LIN {X 0,Y 297.473,Z 181.693,A -85,B 0,C 180,E1 -16448.382,E2 -16448.382} C_VEL
LIN {X 0,Y 297.609,Z 178.436,A -85,B 0,C 180,E1 -16452.122,E2 -16452.122} C_VEL
LIN {X 0,Y 297.859,Z 175.705,A -85,B 0,C 180,E1 -16455.326,E2 -16455.326} C_VEL
LIN {X 0,Y 298.134,Z 175.347,A -85,B 0,C 180,E1 -16457.751,E2 -16457.751} C_VEL
LIN {X 0,Y 298.702,Z 175.277,A -85,B 0,C 180,E1 -16461.884,E2 -16461.884} C_VEL
LIN {X 0,Y 298.65,Z 175.283,A -85,B 0,C 180,E1 -16464.598,E2 -16464.598} C_VEL
LIN {X 0,Y 298.921,Z 175.249,A -85,B 0,C 180,E1 -16468.653,E2 -16468.653} C_VEL
LIN {X 0,Y 298.921,Z 175.247,A -85,B 0,C 180,E1 -16471.347,E2 -16471.347} C_VEL
LIN {X 0,Y 298.794,Z 175.264,A -85,B 0,C 180,E1 -16476.754,E2 -16476.754} C_VEL
LIN {X 0,Y 298.677,Z 175.281,A -85,B 0,C 180,E1 -16479.48,E2 -16479.48} C_VEL
LIN {X 0,Y 298.549,Z 175.299,A -85,B 0,C 180,E1 -16483.615,E2 -16483.615} C_VEL
LIN {X 0,Y 298.545,Z 175.295,A -85,B 0,C 180,E1 -16486.409,E2 -16486.409} C_VEL
LIN {X 0,Y 298.508,Z 175.304,A -85,B 0,C 180,E1 -16489.655,E2 -16489.655} C_VEL
LIN {X 0,Y 298.454,Z 175.31,A -85,B 0,C 180,E1 -16493.598,E2 -16493.598} C_VEL
LIN {X 0,Y 298.482,Z 175.3,A -85,B 0,C 180,E1 -16496.575,E2 -16496.575} C_VEL
LIN {X 0,Y 298.413,Z 175.314,A -85,B 0,C 180,E1 -16499.642,E2 -16499.642} C_VEL
LIN {X 0,Y 298.391,Z 175.315,A -85,B 0,C 180,E1 -16502.801,E2 -16502.801} C_VEL
LIN {X 0,Y 298.441,Z 175.307,A -85,B 0,C 180,E1 -16506.807,E2 -16506.807} C_VEL
LIN {X 0,Y 298.385,Z 175.319,A -85,B 0,C 180,E1 -16511.088,E2 -16511.088} C_VEL
LIN {X 0,Y 298.386,Z 175.318,A -85,B 0,C 180,E1 -16515.042,E2 -16515.042} C_VEL
LIN {X 0,Y 298.385,Z 175.316,A -85,B 0,C 180,E1 -16518.913,E2 -16518.913} C_VEL
LIN {X 0,Y 298.442,Z 175.309,A -85,B 0,C 180,E1 -16523.193,E2 -16523.193} C_VEL
LIN {X 0,Y 298.393,Z 175.314,A -85,B 0,C 180,E1 -16527.2,E2 -16527.2} C_VEL
LIN {X 0,Y 298.425,Z 175.311,A -85,B 0,C 180,E1 -16530.617,E2 -16530.617} C_VEL
LIN {X 0,Y 298.476,Z 175.301,A -85,B 0,C 180,E1 -16533.477,E2 -16533.477} C_VEL
LIN {X 0,Y 298.435,Z 175.312,A -85,B 0,C 180,E1 -16536.698,E2 -16536.698} C_VEL
LIN {X 0,Y 298.539,Z 175.296,A -85,B 0,C 180,E1 -16540.758,E2 -16540.758} C_VEL
LIN {X 0,Y 298.593,Z 175.286,A -85,B 0,C 180,E1 -16544.996,E2 -16544.996} C_VEL
LIN {X 0,Y 298.592,Z 175.288,A -85,B 0,C 180,E1 -16549.147,E2 -16549.147} C_VEL
LIN {X 0,Y 298.741,Z 175.272,A -85,B 0,C 180,E1 -16551.886,E2 -16551.886} C_VEL
LIN {X 0,Y 298.713,Z 175.271,A -85,B 0,C 180,E1 -16553.806,E2 -16553.806} C_VEL
LIN {X 0,Y 297.983,Z 175.364,A -85,B 0,C 180,E1 -16554.931,E2 -16554.931} C_VEL
LIN {X 0,Y 295.181,Z 175.711,A -85,B 0,C 180,E1 -16556.768,E2 -16556.768} C_VEL
LIN {X 0,Y 292.899,Z 175.999,A -85,B 0,C 180,E1 -16558.258,E2 -16558.258} C_VEL
LIN {X 0,Y 291.986,Z 176.11,A -85,B 0,C 180,E1 -16559.41,E2 -16559.41} C_VEL
LIN {X 0,Y 291.944,Z 176.117,A -85,B 0,C 180,E1 -16559.799,E2 -16559.799} C_VEL
LIN {X 0,Y 291.788,Z 176.136,A -85,B 0,C 180,E1 -16562.762,E2 -16562.762} C_VEL
LIN {X 0,Y 291.7,Z 176.146,A -85,B 0,C 180,E1 -16566.92,E2 -16566.92} C_VEL
LIN {X 0,Y 291.569,Z 176.164,A -85,B 0,C 180,E1 -16569.715,E2 -16569.715} C_VEL
LIN {X 0,Y 291.524,Z 176.172,A -85,B 0,C 180,E1 -16573.951,E2 -16573.951} C_VEL
LIN {X 0,Y 291.489,Z 176.172,A -85,B 0,C 180,E1 -16576.818,E2 -16576.818} C_VEL
LIN {X 0,Y 291.452,Z 176.18,A -85,B 0,C 180,E1 -16579.875,E2 -16579.875} C_VEL
LIN {X 0,Y 291.401,Z 176.185,A -85,B 0,C 180,E1 -16584.206,E2 -16584.206} C_VEL
LIN {X 0,Y 291.421,Z 176.186,A -85,B 0,C 180,E1 -16587.272,E2 -16587.272} C_VEL
LIN {X 0,Y 291.336,Z 176.193,A -85,B 0,C 180,E1 -16590.438,E2 -16590.438} C_VEL
LIN {X 0,Y 291.347,Z 176.194,A -85,B 0,C 180,E1 -16593.699,E2 -16593.699} C_VEL
LIN {X 0,Y 291.378,Z 176.192,A -85,B 0,C 180,E1 -16597.255,E2 -16597.255} C_VEL
LIN {X 0,Y 291.382,Z 176.234,A -85,B 0,C 180,E1 -16599.836,E2 -16599.836} C_VEL
LIN {X 0,Y 292.261,Z 181.111,A -85,B 0,C 180,E1 -16603.829,E2 -16603.829} C_VEL
LIN {X 0,Y 293.231,Z 186.36,A -85,B 0,C 180,E1 -16607.849,E2 -16607.849} C_VEL
LIN {X 0,Y 294.105,Z 191.57,A -85,B 0,C 180,E1 -16611.589,E2 -16611.589} C_VEL
LIN {X 0,Y 294.167,Z 194.116,A -85,B 0,C 180,E1 -16613.325,E2 -16613.325} C_VEL
LIN {X 0,Y 293.464,Z 199.141,A -85,B 0,C 180,E1 -16616.577,E2 -16616.577} C_VEL
LIN {X 0,Y 292.415,Z 205.473,A -85,B 0,C 180,E1 -16620.549,E2 -16620.549} C_VEL
LIN {X 0,Y 291.542,Z 211.574,A -85,B 0,C 180,E1 -16624.284,E2 -16624.284} C_VEL
LIN {X 0,Y 291.27,Z 214.004,A -85,B 0,C 180,E1 -16625.724,E2 -16625.724} C_VEL
LIN {X 0,Y 293.669,Z 227.805,A -85,B 0,C 180,E1 -16626.542,E2 -16626.542} C_VEL
LIN {X 0,Y 295.547,Z 241.488,A -85,B 0,C 180,E1 -16627.637,E2 -16627.637} C_VEL
LIN {X 0,Y 296.631,Z 253.134,A -85,B 0,C 180,E1 -16628.799,E2 -16628.799} C_VEL
LIN {X 0,Y 296.996,Z 262.647,A -85,B 0,C 180,E1 -16629.933,E2 -16629.933} C_VEL
LIN {X 0,Y 295.444,Z 272.588,A -85,B 0,C 180,E1 -16631.268,E2 -16631.268} C_VEL
LIN {X 0,Y 293.939,Z 283.435,A -85,B 0,C 180,E1 -16633.114,E2 -16633.114} C_VEL
LIN {X 0,Y 292.546,Z 292.482,A -85,B 0,C 180,E1 -16635.034,E2 -16635.034} C_VEL
LIN {X 0,Y 291.363,Z 300.313,A -85,B 0,C 180,E1 -16637.108,E2 -16637.108} C_VEL
LIN {X 0,Y 290.452,Z 307.494,A -85,B 0,C 180,E1 -16639.544,E2 -16639.544} C_VEL
LIN {X 0,Y 289.911,Z 312.271,A -85,B 0,C 180,E1 -16641.637,E2 -16641.637} C_VEL
LIN {X 0,Y 289.677,Z 316.494,A -85,B 0,C 180,E1 -16644.117,E2 -16644.117} C_VEL
LIN {X 0,Y 289.602,Z 318.523,A -85,B 0,C 180,E1 -16645.825,E2 -16645.825} C_VEL
LIN {X 0,Y 289.558,Z 319.73,A -85,B 0,C 180,E1 -16647.218,E2 -16647.218} C_VEL
LIN {X 0,Y 289.58,Z 320.506,A -85,B 0,C 180,E1 -16648.61,E2 -16648.61} C_VEL
LIN {X 0,Y 289.688,Z 320.856,A -85,B 0,C 180,E1 -16650,E2 -16650} C_VEL
LIN {X 0,Y 289.545,Z 320.344,A -85,B 0,C 180,E1 -16652.783,E2 -16652.783} C_VEL
LIN {X 0,Y 289.557,Z 319.479,A -85,B 0,C 180,E1 -16654.176,E2 -16654.176} C_VEL
LIN {X 0,Y 289.633,Z 317.927,A -85,B 0,C 180,E1 -16655.798,E2 -16655.798} C_VEL
LIN {X 0,Y 289.908,Z 314.345,A -85,B 0,C 180,E1 -16658.364,E2 -16658.364} C_VEL
LIN {X 0,Y 290.452,Z 310.262,A -85,B 0,C 180,E1 -16660.456,E2 -16660.456} C_VEL
LIN {X 0,Y 291.439,Z 304.066,A -85,B 0,C 180,E1 -16662.889,E2 -16662.889} C_VEL
LIN {X 0,Y 292.984,Z 296.118,A -85,B 0,C 180,E1 -16665.3,E2 -16665.3} C_VEL
LIN {X 0,Y 294.468,Z 288.574,A -85,B 0,C 180,E1 -16667.128,E2 -16667.128} C_VEL
LIN {X 0,Y 296.202,Z 278.852,A -85,B 0,C 180,E1 -16669.041,E2 -16669.041} C_VEL
LIN {X 0,Y 298.212,Z 268.241,A -85,B 0,C 180,E1 -16670.702,E2 -16670.702} C_VEL
LIN {X 0,Y 298.925,Z 263.295,A -85,B 0,C 180,E1 -16671.372,E2 -16671.372} C_VEL
LIN {X 0,Y 298.806,Z 251.482,A -85,B 0,C 180,E1 -16672.872,E2 -16672.872} C_VEL
LIN {X 0,Y 297.979,Z 239.718,A -85,B 0,C 180,E1 -16674.143,E2 -16674.143} C_VEL
LIN {X 0,Y 295.872,Z 227.27,A -85,B 0,C 180,E1 -16675.344,E2 -16675.344} C_VEL
LIN {X 0,Y 292.582,Z 214.464,A -85,B 0,C 180,E1 -16676.448,E2 -16676.448} C_VEL
LIN {X 0,Y 291.854,Z 211.366,A -85,B 0,C 180,E1 -16676.694,E2 -16676.694} C_VEL
LIN {X 0,Y 292.741,Z 205.794,A -85,B 0,C 180,E1 -16680.276,E2 -16680.276} C_VEL
LIN {X 0,Y 293.888,Z 199.966,A -85,B 0,C 180,E1 -16684.193,E2 -16684.193} C_VEL
LIN {X 0,Y 294.505,Z 196.544,A -85,B 0,C 180,E1 -16686.627,E2 -16686.627} C_VEL
LIN {X 0,Y 294.392,Z 193.2,A -85,B 0,C 180,E1 -16689.234,E2 -16689.234} C_VEL
LIN {X 0,Y 293.627,Z 188.721,A -85,B 0,C 180,E1 -16693.112,E2 -16693.112} C_VEL
LIN {X 0,Y 293.064,Z 185.716,A -85,B 0,C 180,E1 -16696.008,E2 -16696.008} C_VEL
LIN {X 0,Y 292.457,Z 182.486,A -85,B 0,C 180,E1 -16699.545,E2 -16699.545} C_VEL
LIN {X 0,Y 292.058,Z 179.712,A -85,B 0,C 180,E1 -16703.015,E2 -16703.015} C_VEL
LIN {X 0,Y 291.588,Z 177.48,A -85,B 0,C 180,E1 -16706.333,E2 -16706.333} C_VEL
LIN {X 0,Y 291.4,Z 176.52,A -85,B 0,C 180,E1 -16707.953,E2 -16707.953} C_VEL
LIN {X 0,Y 291.381,Z 176.187,A -85,B 0,C 180,E1 -16711.158,E2 -16711.158} C_VEL
LIN {X 0,Y 291.419,Z 176.187,A -85,B 0,C 180,E1 -16714.271,E2 -16714.271} C_VEL
LIN {X 0,Y 291.385,Z 176.186,A -85,B 0,C 180,E1 -16717.299,E2 -16717.299} C_VEL
LIN {X 0,Y 291.462,Z 176.177,A -85,B 0,C 180,E1 -16720.27,E2 -16720.27} C_VEL
LIN {X 0,Y 291.501,Z 176.175,A -85,B 0,C 180,E1 -16724.665,E2 -16724.665} C_VEL
LIN {X 0,Y 291.541,Z 176.171,A -85,B 0,C 180,E1 -16728.88,E2 -16728.88} C_VEL
LIN {X 0,Y 291.713,Z 176.149,A -85,B 0,C 180,E1 -16731.688,E2 -16731.688} C_VEL
LIN {X 0,Y 291.635,Z 176.159,A -85,B 0,C 180,E1 -16734.468,E2 -16734.468} C_VEL
LIN {X 0,Y 291.894,Z 176.128,A -85,B 0,C 180,E1 -16738.62,E2 -16738.62} C_VEL
LIN {X 0,Y 291.894,Z 176.126,A -85,B 0,C 180,E1 -16741.379,E2 -16741.379} C_VEL
LIN {X 0,Y 291.752,Z 177.229,A -85,B 0,C 180,E1 -16744.143,E2 -16744.143} C_VEL
LIN {X 0,Y 292.061,Z 178.577,A -85,B 0,C 180,E1 -16746.91,E2 -16746.91} C_VEL
LIN {X 0,Y 291.978,Z 180.14,A -85,B 0,C 180,E1 -16749.699,E2 -16749.699} C_VEL
LIN {X 0,Y 291.787,Z 181.835,A -85,B 0,C 180,E1 -16752.519,E2 -16752.519} C_VEL
LIN {X 0,Y 291.378,Z 184.632,A -85,B 0,C 180,E1 -16756.824,E2 -16756.824} C_VEL
LIN {X 0,Y 291.273,Z 185.686,A -85,B 0,C 180,E1 -16758.371,E2 -16758.371} C_VEL
LIN {X 0,Y 292.352,Z 188.722,A -85,B 0,C 180,E1 -16758.664,E2 -16758.664} C_VEL
LIN {X 0,Y 296.964,Z 200.311,A -85,B 0,C 180,E1 -16759.952,E2 -16759.952} C_VEL
LIN {X 0,Y 300.069,Z 210.537,A -85,B 0,C 180,E1 -16761.167,E2 -16761.167} C_VEL
LIN {X 0,Y 302.406,Z 221.365,A -85,B 0,C 180,E1 -16762.548,E2 -16762.548} C_VEL
LIN {X 0,Y 302.217,Z 224.598,A -85,B 0,C 180,E1 -16762.924,E2 -16762.924} C_VEL
LIN {X 0,Y 300.369,Z 236.248,A -85,B 0,C 180,E1 -16764.371,E2 -16764.371} C_VEL
LIN {X 0,Y 298.483,Z 247.026,A -85,B 0,C 180,E1 -16766.094,E2 -16766.094} C_VEL
LIN {X 0,Y 296.667,Z 256.099,A -85,B 0,C 180,E1 -16767.896,E2 -16767.896} C_VEL
LIN {X 0,Y 294.899,Z 264.601,A -85,B 0,C 180,E1 -16770.03,E2 -16770.03} C_VEL
LIN {X 0,Y 293.209,Z 271.816,A -85,B 0,C 180,E1 -16772.325,E2 -16772.325} C_VEL
LIN {X 0,Y 292.129,Z 276.595,A -85,B 0,C 180,E1 -16774.287,E2 -16774.287} C_VEL
LIN {X 0,Y 291.332,Z 280.279,A -85,B 0,C 180,E1 -16776.229,E2 -16776.229} C_VEL
LIN {X 0,Y 290.401,Z 283.973,A -85,B 0,C 180,E1 -16778.992,E2 -16778.992} C_VEL
LIN {X 0,Y 289.859,Z 285.745,A -85,B 0,C 180,E1 -16781.267,E2 -16781.267} C_VEL
LIN {X 0,Y 289.616,Z 286.413,A -85,B 0,C 180,E1 -16783.281,E2 -16783.281} C_VEL
LIN {X 0,Y 289.521,Z 286.258,A -85,B 0,C 180,E1 -16785.254,E2 -16785.254} C_VEL
LIN {X 0,Y 289.563,Z 285.285,A -85,B 0,C 180,E1 -16787.188,E2 -16787.188} C_VEL
LIN {X 0,Y 289.829,Z 283.546,A -85,B 0,C 180,E1 -16789.101,E2 -16789.101} C_VEL
LIN {X 0,Y 290.2,Z 281.076,A -85,B 0,C 180,E1 -16790.974,E2 -16790.974} C_VEL
LIN {X 0,Y 290.658,Z 277.615,A -85,B 0,C 180,E1 -16792.931,E2 -16792.931} C_VEL
LIN {X 0,Y 291.355,Z 272.592,A -85,B 0,C 180,E1 -16795.098,E2 -16795.098} C_VEL
LIN {X 0,Y 292.279,Z 266.034,A -85,B 0,C 180,E1 -16797.307,E2 -16797.307} C_VEL
LIN {X 0,Y 293.374,Z 258.821,A -85,B 0,C 180,E1 -16799.251,E2 -16799.251} C_VEL
LIN {X 0,Y 294.688,Z 250.261,A -85,B 0,C 180,E1 -16801.122,E2 -16801.122} C_VEL
LIN {X 0,Y 296.086,Z 239.523,A -85,B 0,C 180,E1 -16803.002,E2 -16803.002} C_VEL
LIN {X 0,Y 297.431,Z 229.141,A -85,B 0,C 180,E1 -16804.457,E2 -16804.457} C_VEL
LIN {X 0,Y 298.727,Z 217.214,A -85,B 0,C 180,E1 -16805.78,E2 -16805.78} C_VEL
LIN {X 0,Y 297.949,Z 211.851,A -85,B 0,C 180,E1 -16806.359,E2 -16806.359} C_VEL
LIN {X 0,Y 295.508,Z 200.646,A -85,B 0,C 180,E1 -16807.449,E2 -16807.449} C_VEL
LIN {X 0,Y 292.062,Z 188.008,A -85,B 0,C 180,E1 -16808.471,E2 -16808.471} C_VEL
LIN {X 0,Y 290.437,Z 182.117,A -85,B 0,C 180,E1 -16808.856,E2 -16808.856} C_VEL
LIN {X 0,Y 290.636,Z 178.451,A -85,B 0,C 180,E1 -16813.131,E2 -16813.131} C_VEL
LIN {X 0,Y 290.867,Z 176.256,A -85,B 0,C 180,E1 -16816.017,E2 -16816.017} C_VEL
LIN {X 0,Y 291.428,Z 176.186,A -85,B 0,C 180,E1 -16820.281,E2 -16820.281} C_VEL
LIN {X 0,Y 291.716,Z 176.146,A -85,B 0,C 180,E1 -16823.081,E2 -16823.081} C_VEL
LIN {X 0,Y 291.887,Z 176.125,A -85,B 0,C 180,E1 -16828.62,E2 -16828.62} C_VEL
LIN {X 0,Y 291.887,Z 176.124,A -85,B 0,C 180,E1 -16831.379,E2 -16831.379} C_VEL
LIN {X 0,Y 291.743,Z 176.142,A -85,B 0,C 180,E1 -16836.918,E2 -16836.918} C_VEL
LIN {X 0,Y 291.626,Z 176.161,A -85,B 0,C 180,E1 -16839.712,E2 -16839.712} C_VEL
LIN {X 0,Y 291.519,Z 176.174,A -85,B 0,C 180,E1 -16843.95,E2 -16843.95} C_VEL
LIN {X 0,Y 291.484,Z 176.174,A -85,B 0,C 180,E1 -16846.818,E2 -16846.818} C_VEL
LIN {X 0,Y 291.447,Z 176.182,A -85,B 0,C 180,E1 -16849.875,E2 -16849.875} C_VEL
LIN {X 0,Y 291.396,Z 176.185,A -85,B 0,C 180,E1 -16854.205,E2 -16854.205} C_VEL
LIN {X 0,Y 291.415,Z 176.184,A -85,B 0,C 180,E1 -16857.272,E2 -16857.272} C_VEL
LIN {X 0,Y 291.331,Z 176.193,A -85,B 0,C 180,E1 -16860.437,E2 -16860.437} C_VEL
LIN {X 0,Y 291.341,Z 176.193,A -85,B 0,C 180,E1 -16863.699,E2 -16863.699} C_VEL
LIN {X 0,Y 291.369,Z 176.19,A -85,B 0,C 180,E1 -16867.253,E2 -16867.253} C_VEL
LIN {X 0,Y 291.33,Z 176.194,A -85,B 0,C 180,E1 -16870.643,E2 -16870.643} C_VEL
LIN {X 0,Y 291.311,Z 176.196,A -85,B 0,C 180,E1 -16874.398,E2 -16874.398} C_VEL
LIN {X 0,Y 291.324,Z 176.191,A -85,B 0,C 180,E1 -16878.405,E2 -16878.405} C_VEL
LIN {X 0,Y 291.345,Z 176.193,A -85,B 0,C 180,E1 -16881.158,E2 -16881.158} C_VEL
LIN {X 0,Y 291.359,Z 176.193,A -85,B 0,C 180,E1 -16884.627,E2 -16884.627} C_VEL
LIN {X 0,Y 291.368,Z 176.187,A -85,B 0,C 180,E1 -16887.951,E2 -16887.951} C_VEL
LIN {X 0,Y 291.375,Z 176.185,A -85,B 0,C 180,E1 -16891.158,E2 -16891.158} C_VEL
LIN {X 0,Y 291.411,Z 176.183,A -85,B 0,C 180,E1 -16894.272,E2 -16894.272} C_VEL
LIN {X 0,Y 291.388,Z 176.186,A -85,B 0,C 180,E1 -16897.301,E2 -16897.301} C_VEL
LIN {X 0,Y 291.458,Z 176.18,A -85,B 0,C 180,E1 -16900.271,E2 -16900.271} C_VEL
LIN {X 0,Y 291.555,Z 176.165,A -85,B 0,C 180,E1 -16904.624,E2 -16904.624} C_VEL
LIN {X 0,Y 291.536,Z 176.168,A -85,B 0,C 180,E1 -16908.881,E2 -16908.881} C_VEL
LIN {X 0,Y 291.688,Z 176.15,A -85,B 0,C 180,E1 -16911.689,E2 -16911.689} C_VEL
LIN {X 0,Y 291.628,Z 176.157,A -85,B 0,C 180,E1 -16914.469,E2 -16914.469} C_VEL
LIN {X 0,Y 291.89,Z 176.122,A -85,B 0,C 180,E1 -16918.621,E2 -16918.621} C_VEL
LIN {X 0,Y 291.944,Z 176.117,A -85,B 0,C 180,E1 -16919.799,E2 -16919.799} C_VEL
LIN {X 0,Y 291.324,Z 176.203,A -85,B 0,C 180,E1 -16920.948,E2 -16920.948} C_VEL
LIN {X 0,Y 288.343,Z 176.58,A -85,B 0,C 180,E1 -16922.813,E2 -16922.813} C_VEL
LIN {X 0,Y 285.768,Z 176.896,A -85,B 0,C 180,E1 -16924.328,E2 -16924.328} C_VEL
LIN {X 0,Y 284.666,Z 177.027,A -85,B 0,C 180,E1 -16925.506,E2 -16925.506} C_VEL
LIN {X 0,Y 284.582,Z 177.034,A -85,B 0,C 180,E1 -16925.906,E2 -16925.906} C_VEL
LIN {X 0,Y 284.616,Z 177.026,A -85,B 0,C 180,E1 -16928.99,E2 -16928.99} C_VEL
LIN {X 0,Y 284.477,Z 177.047,A -85,B 0,C 180,E1 -16932.848,E2 -16932.848} C_VEL
LIN {X 0,Y 284.489,Z 177.049,A -85,B 0,C 180,E1 -16935.769,E2 -16935.769} C_VEL
LIN {X 0,Y 284.382,Z 177.059,A -85,B 0,C 180,E1 -16940.243,E2 -16940.243} C_VEL
LIN {X 0,Y 284.371,Z 177.062,A -85,B 0,C 180,E1 -16943.876,E2 -16943.876} C_VEL
LIN {X 0,Y 284.396,Z 177.06,A -85,B 0,C 180,E1 -16947.173,E2 -16947.173} C_VEL
LIN {X 0,Y 284.296,Z 177.074,A -85,B 0,C 180,E1 -16951.275,E2 -16951.275} C_VEL
LIN {X 0,Y 284.343,Z 177.068,A -85,B 0,C 180,E1 -16955.349,E2 -16955.349} C_VEL
LIN {X 0,Y 284.362,Z 177.234,A -85,B 0,C 180,E1 -16959.526,E2 -16959.526} C_VEL
LIN {X 0,Y 285.227,Z 182.114,A -85,B 0,C 180,E1 -16963.625,E2 -16963.625} C_VEL
LIN {X 0,Y 286.136,Z 187.021,A -85,B 0,C 180,E1 -16967.465,E2 -16967.465} C_VEL
LIN {X 0,Y 286.875,Z 190.986,A -85,B 0,C 180,E1 -16970.435,E2 -16970.435} C_VEL
LIN {X 0,Y 287.141,Z 194.822,A -85,B 0,C 180,E1 -16973.156,E2 -16973.156} C_VEL
LIN {X 0,Y 286.698,Z 198.598,A -85,B 0,C 180,E1 -16975.68,E2 -16975.68} C_VEL
LIN {X 0,Y 285.64,Z 204.418,A -85,B 0,C 180,E1 -16979.447,E2 -16979.447} C_VEL
LIN {X 0,Y 284.621,Z 211.01,A -85,B 0,C 180,E1 -16983.611,E2 -16983.611} C_VEL
LIN {X 0,Y 284.292,Z 213.57,A -85,B 0,C 180,E1 -16985.208,E2 -16985.208} C_VEL
LIN {X 0,Y 286.616,Z 227.014,A -85,B 0,C 180,E1 -16986.017,E2 -16986.017} C_VEL
LIN {X 0,Y 288.416,Z 239.822,A -85,B 0,C 180,E1 -16987.053,E2 -16987.053} C_VEL
LIN {X 0,Y 289.601,Z 252.402,A -85,B 0,C 180,E1 -16988.328,E2 -16988.328} C_VEL
LIN {X 0,Y 290.103,Z 262.902,A -85,B 0,C 180,E1 -16989.62,E2 -16989.62} C_VEL
LIN {X 0,Y 288.36,Z 273.793,A -85,B 0,C 180,E1 -16991.16,E2 -16991.16} C_VEL
LIN {X 0,Y 286.926,Z 283.608,A -85,B 0,C 180,E1 -16992.907,E2 -16992.907} C_VEL
LIN {X 0,Y 285.66,Z 291.673,A -85,B 0,C 180,E1 -16994.664,E2 -16994.664} C_VEL
LIN {X 0,Y 284.425,Z 299.597,A -85,B 0,C 180,E1 -16996.788,E2 -16996.788} C_VEL
LIN {X 0,Y 283.646,Z 304.963,A -85,B 0,C 180,E1 -16998.567,E2 -16998.567} C_VEL
LIN {X 0,Y 283.042,Z 310.211,A -85,B 0,C 180,E1 -17000.712,E2 -17000.712} C_VEL
LIN {X 0,Y 282.666,Z 314.267,A -85,B 0,C 180,E1 -17002.859,E2 -17002.859} C_VEL
LIN {X 0,Y 282.569,Z 316.36,A -85,B 0,C 180,E1 -17004.291,E2 -17004.291} C_VEL
LIN {X 0,Y 282.522,Z 318.006,A -85,B 0,C 180,E1 -17005.72,E2 -17005.72} C_VEL
LIN {X 0,Y 282.485,Z 319.235,A -85,B 0,C 180,E1 -17007.148,E2 -17007.148} C_VEL
LIN {X 0,Y 282.495,Z 320.049,A -85,B 0,C 180,E1 -17008.575,E2 -17008.575} C_VEL
LIN {X 0,Y 282.599,Z 320.42,A -85,B 0,C 180,E1 -17010,E2 -17010} C_VEL
LIN {X 0,Y 282.471,Z 319.946,A -85,B 0,C 180,E1 -17012.853,E2 -17012.853} C_VEL
LIN {X 0,Y 282.459,Z 319.113,A -85,B 0,C 180,E1 -17014.281,E2 -17014.281} C_VEL
LIN {X 0,Y 282.525,Z 317.834,A -85,B 0,C 180,E1 -17015.711,E2 -17015.711} C_VEL
LIN {X 0,Y 282.871,Z 314.053,A -85,B 0,C 180,E1 -17018.573,E2 -17018.573} C_VEL
LIN {X 0,Y 283.431,Z 310.028,A -85,B 0,C 180,E1 -17020.718,E2 -17020.718} C_VEL
LIN {X 0,Y 284.284,Z 304.895,A -85,B 0,C 180,E1 -17022.856,E2 -17022.856} C_VEL
LIN {X 0,Y 285.654,Z 298.513,A -85,B 0,C 180,E1 -17024.972,E2 -17024.972} C_VEL
LIN {X 0,Y 287.278,Z 290.595,A -85,B 0,C 180,E1 -17027.072,E2 -17027.072} C_VEL
LIN {X 0,Y 289.116,Z 280.821,A -85,B 0,C 180,E1 -17029.158,E2 -17029.158} C_VEL
LIN {X 0,Y 291.155,Z 270.809,A -85,B 0,C 180,E1 -17030.858,E2 -17030.858} C_VEL
LIN {X 0,Y 292.22,Z 264.91,A -85,B 0,C 180,E1 -17031.702,E2 -17031.702} C_VEL
LIN {X 0,Y 292.276,Z 252.503,A -85,B 0,C 180,E1 -17033.377,E2 -17033.377} C_VEL
LIN {X 0,Y 291.592,Z 241.508,A -85,B 0,C 180,E1 -17034.642,E2 -17034.642} C_VEL
LIN {X 0,Y 289.649,Z 229.307,A -85,B 0,C 180,E1 -17035.897,E2 -17035.897} C_VEL
LIN {X 0,Y 286.682,Z 217.022,A -85,B 0,C 180,E1 -17037.046,E2 -17037.046} C_VEL
LIN {X 0,Y 285.078,Z 211.471,A -85,B 0,C 180,E1 -17037.524,E2 -17037.524} C_VEL
LIN {X 0,Y 285.022,Z 210.856,A -85,B 0,C 180,E1 -17037.589,E2 -17037.589} C_VEL
LIN {X 0,Y 286.189,Z 204.454,A -85,B 0,C 180,E1 -17041.869,E2 -17041.869} C_VEL
LIN {X 0,Y 287.126,Z 199.845,A -85,B 0,C 180,E1 -17045.115,E2 -17045.115} C_VEL
LIN {X 0,Y 287.53,Z 196.46,A -85,B 0,C 180,E1 -17047.667,E2 -17047.667} C_VEL
LIN {X 0,Y 287.139,Z 192.9,A -85,B 0,C 180,E1 -17050.645,E2 -17050.645} C_VEL
LIN {X 0,Y 286.638,Z 189.94,A -85,B 0,C 180,E1 -17053.356,E2 -17053.356} C_VEL
LIN {X 0,Y 285.871,Z 185.854,A -85,B 0,C 180,E1 -17057.522,E2 -17057.522} C_VEL
LIN {X 0,Y 285.492,Z 183.577,A -85,B 0,C 180,E1 -17060.204,E2 -17060.204} C_VEL
LIN {X 0,Y 285.014,Z 180.891,A -85,B 0,C 180,E1 -17063.714,E2 -17063.714} C_VEL
LIN {X 0,Y 284.589,Z 178.723,A -85,B 0,C 180,E1 -17067.103,E2 -17067.103} C_VEL
LIN {X 0,Y 284.359,Z 177.065,A -85,B 0,C 180,E1 -17070.375,E2 -17070.375} C_VEL
LIN {X 0,Y 284.38,Z 177.059,A -85,B 0,C 180,E1 -17073.586,E2 -17073.586} C_VEL
LIN {X 0,Y 284.371,Z 177.063,A -85,B 0,C 180,E1 -17076.707,E2 -17076.707} C_VEL
LIN {X 0,Y 284.39,Z 177.059,A -85,B 0,C 180,E1 -17081.26,E2 -17081.26} C_VEL
LIN {X 0,Y 284.467,Z 177.051,A -85,B 0,C 180,E1 -17085.696,E2 -17085.696} C_VEL
LIN {X 0,Y 284.57,Z 177.039,A -85,B 0,C 180,E1 -17090.044,E2 -17090.044} C_VEL
LIN {X 0,Y 284.703,Z 177.022,A -85,B 0,C 180,E1 -17092.909,E2 -17092.909} C_VEL
LIN {X 0,Y 284.86,Z 177.004,A -85,B 0,C 180,E1 -17098.586,E2 -17098.586} C_VEL
LIN {X 0,Y 284.94,Z 176.993,A -85,B 0,C 180,E1 -17099.999,E2 -17099.999} C_VEL
LIN {X 0,Y 284.908,Z 178.004,A -85,B 0,C 180,E1 -17102.827,E2 -17102.827} C_VEL
LIN {X 0,Y 285.086,Z 180.013,A -85,B 0,C 180,E1 -17107.08,E2 -17107.08} C_VEL
LIN {X 0,Y 284.96,Z 181.565,A -85,B 0,C 180,E1 -17109.941,E2 -17109.941} C_VEL
LIN {X 0,Y 284.749,Z 183.277,A -85,B 0,C 180,E1 -17112.834,E2 -17112.834} C_VEL
LIN {X 0,Y 284.341,Z 186.086,A -85,B 0,C 180,E1 -17117.253,E2 -17117.253} C_VEL
LIN {X 0,Y 284.316,Z 186.211,A -85,B 0,C 180,E1 -17117.44,E2 -17117.44} C_VEL
LIN {X 0,Y 285.44,Z 189.331,A -85,B 0,C 180,E1 -17117.785,E2 -17117.785} C_VEL
LIN {X 0,Y 289.629,Z 199.309,A -85,B 0,C 180,E1 -17118.984,E2 -17118.984} C_VEL
LIN {X 0,Y 293.173,Z 210.255,A -85,B 0,C 180,E1 -17120.34,E2 -17120.34} C_VEL
LIN {X 0,Y 295.483,Z 220.547,A -85,B 0,C 180,E1 -17121.706,E2 -17121.706} C_VEL
LIN {X 0,Y 296.053,Z 224.104,A -85,B 0,C 180,E1 -17122.207,E2 -17122.207} C_VEL
LIN {X 0,Y 294.229,Z 235.254,A -85,B 0,C 180,E1 -17123.583,E2 -17123.583} C_VEL
LIN {X 0,Y 292.458,Z 245.222,A -85,B 0,C 180,E1 -17125.136,E2 -17125.136} C_VEL
LIN {X 0,Y 290.481,Z 254.563,A -85,B 0,C 180,E1 -17126.942,E2 -17126.942} C_VEL
LIN {X 0,Y 288.775,Z 262.385,A -85,B 0,C 180,E1 -17128.819,E2 -17128.819} C_VEL
LIN {X 0,Y 287.037,Z 269.76,A -85,B 0,C 180,E1 -17131.022,E2 -17131.022} C_VEL
LIN {X 0,Y 285.613,Z 275.476,A -85,B 0,C 180,E1 -17133.214,E2 -17133.214} C_VEL
LIN {X 0,Y 284.597,Z 279.9,A -85,B 0,C 180,E1 -17135.42,E2 -17135.42} C_VEL
LIN {X 0,Y 283.727,Z 283.107,A -85,B 0,C 180,E1 -17137.566,E2 -17137.566} C_VEL
LIN {X 0,Y 282.979,Z 285.674,A -85,B 0,C 180,E1 -17140.219,E2 -17140.219} C_VEL
LIN {X 0,Y 282.664,Z 286.644,A -85,B 0,C 180,E1 -17142.167,E2 -17142.167} C_VEL
LIN {X 0,Y 282.485,Z 286.878,A -85,B 0,C 180,E1 -17144.155,E2 -17144.155} C_VEL
LIN {X 0,Y 282.427,Z 286.294,A -85,B 0,C 180,E1 -17146.189,E2 -17146.189} C_VEL
LIN {X 0,Y 282.599,Z 284.843,A -85,B 0,C 180,E1 -17148.25,E2 -17148.25} C_VEL
LIN {X 0,Y 282.98,Z 282.479,A -85,B 0,C 180,E1 -17150.344,E2 -17150.344} C_VEL
LIN {X 0,Y 283.466,Z 279.044,A -85,B 0,C 180,E1 -17152.501,E2 -17152.501} C_VEL
LIN {X 0,Y 284.122,Z 274.362,A -85,B 0,C 180,E1 -17154.713,E2 -17154.713} C_VEL
LIN {X 0,Y 285.113,Z 267.611,A -85,B 0,C 180,E1 -17157.159,E2 -17157.159} C_VEL
LIN {X 0,Y 286.257,Z 260.303,A -85,B 0,C 180,E1 -17159.236,E2 -17159.236} C_VEL
LIN {X 0,Y 287.608,Z 251.863,A -85,B 0,C 180,E1 -17161.175,E2 -17161.175} C_VEL
LIN {X 0,Y 289.001,Z 241.958,A -85,B 0,C 180,E1 -17163.016,E2 -17163.016} C_VEL
LIN {X 0,Y 290.323,Z 231.668,A -85,B 0,C 180,E1 -17164.552,E2 -17164.552} C_VEL
LIN {X 0,Y 291.754,Z 219.565,A -85,B 0,C 180,E1 -17165.992,E2 -17165.992} C_VEL
LIN {X 0,Y 291.956,Z 217.796,A -85,B 0,C 180,E1 -17166.167,E2 -17166.167} C_VEL
LIN {X 0,Y 289.837,Z 206.676,A -85,B 0,C 180,E1 -17167.379,E2 -17167.379} C_VEL
LIN {X 0,Y 286.832,Z 194.615,A -85,B 0,C 180,E1 -17168.483,E2 -17168.483} C_VEL
LIN {X 0,Y 283.402,Z 182.48,A -85,B 0,C 180,E1 -17169.4,E2 -17169.4} C_VEL
LIN {X 0,Y 283.547,Z 179.71,A -85,B 0,C 180,E1 -17172.696,E2 -17172.696} C_VEL
LIN {X 0,Y 283.773,Z 177.259,A -85,B 0,C 180,E1 -17175.66,E2 -17175.66} C_VEL
LIN {X 0,Y 284.345,Z 177.067,A -85,B 0,C 180,E1 -17180.037,E2 -17180.037} C_VEL
LIN {X 0,Y 284.664,Z 177.025,A -85,B 0,C 180,E1 -17182.909,E2 -17182.909} C_VEL
LIN {X 0,Y 284.853,Z 177.002,A -85,B 0,C 180,E1 -17188.586,E2 -17188.586} C_VEL
LIN {X 0,Y 284.853,Z 177,A -85,B 0,C 180,E1 -17191.414,E2 -17191.414} C_VEL
LIN {X 0,Y 284.695,Z 177.021,A -85,B 0,C 180,E1 -17197.09,E2 -17197.09} C_VEL
LIN {X 0,Y 284.563,Z 177.039,A -85,B 0,C 180,E1 -17199.955,E2 -17199.955} C_VEL
LIN {X 0,Y 284.478,Z 177.049,A -85,B 0,C 180,E1 -17204.303,E2 -17204.303} C_VEL
LIN {X 0,Y 284.422,Z 177.056,A -85,B 0,C 180,E1 -17207.248,E2 -17207.248} C_VEL
LIN {X 0,Y 284.377,Z 177.061,A -85,B 0,C 180,E1 -17210.242,E2 -17210.242} C_VEL
LIN {X 0,Y 284.366,Z 177.063,A -85,B 0,C 180,E1 -17213.875,E2 -17213.875} C_VEL
LIN {X 0,Y 284.391,Z 177.058,A -85,B 0,C 180,E1 -17217.173,E2 -17217.173} C_VEL
LIN {X 0,Y 284.29,Z 177.075,A -85,B 0,C 180,E1 -17221.275,E2 -17221.275} C_VEL
LIN {X 0,Y 284.337,Z 177.065,A -85,B 0,C 180,E1 -17225.348,E2 -17225.348} C_VEL
LIN {X 0,Y 284.305,Z 177.066,A -85,B 0,C 180,E1 -17228.17,E2 -17228.17} C_VEL
LIN {X 0,Y 284.266,Z 177.073,A -85,B 0,C 180,E1 -17232.125,E2 -17232.125} C_VEL
LIN {X 0,Y 284.265,Z 177.071,A -85,B 0,C 180,E1 -17236.192,E2 -17236.192} C_VEL
LIN {X 0,Y 284.304,Z 177.066,A -85,B 0,C 180,E1 -17240.025,E2 -17240.025} C_VEL
LIN {X 0,Y 284.328,Z 177.065,A -85,B 0,C 180,E1 -17243.614,E2 -17243.614} C_VEL
LIN {X 0,Y 284.305,Z 177.068,A -85,B 0,C 180,E1 -17247.19,E2 -17247.19} C_VEL
LIN {X 0,Y 284.354,Z 177.061,A -85,B 0,C 180,E1 -17250.376,E2 -17250.376} C_VEL
LIN {X 0,Y 284.373,Z 177.057,A -85,B 0,C 180,E1 -17253.587,E2 -17253.587} C_VEL
LIN {X 0,Y 284.368,Z 177.064,A -85,B 0,C 180,E1 -17256.708,E2 -17256.708} C_VEL
LIN {X 0,Y 284.403,Z 177.054,A -85,B 0,C 180,E1 -17261.262,E2 -17261.262} C_VEL
LIN {X 0,Y 284.492,Z 177.044,A -85,B 0,C 180,E1 -17264.46,E2 -17264.46} C_VEL
LIN {X 0,Y 284.488,Z 177.047,A -85,B 0,C 180,E1 -17268.602,E2 -17268.602} C_VEL
LIN {X 0,Y 284.639,Z 177.027,A -85,B 0,C 180,E1 -17271.481,E2 -17271.481} C_VEL
LIN {X 0,Y 284.598,Z 177.033,A -85,B 0,C 180,E1 -17274.332,E2 -17274.332} C_VEL
LIN {X 0,Y 284.856,Z 176.998,A -85,B 0,C 180,E1 -17278.587,E2 -17278.587} C_VEL
LIN {X 0,Y 284.855,Z 177,A -85,B 0,C 180,E1 -17281.414,E2 -17281.414} C_VEL
LIN {X 0,Y 284.582,Z 177.034,A -85,B 0,C 180,E1 -17285.906,E2 -17285.906} C_VEL
LIN {X 0,Y 283.921,Z 177.116,A -85,B 0,C 180,E1 -17287.088,E2 -17287.088} C_VEL
LIN {X 0,Y 281.038,Z 177.473,A -85,B 0,C 180,E1 -17289.01,E2 -17289.01} C_VEL
LIN {X 0,Y 278.572,Z 177.784,A -85,B 0,C 180,E1 -17290.572,E2 -17290.572} C_VEL
LIN {X 0,Y 277.5,Z 177.919,A -85,B 0,C 180,E1 -17291.783,E2 -17291.783} C_VEL
LIN {X 0,Y 277.406,Z 177.927,A -85,B 0,C 180,E1 -17292.194,E2 -17292.194} C_VEL
LIN {X 0,Y 277.408,Z 177.927,A -85,B 0,C 180,E1 -17296.182,E2 -17296.182} C_VEL
LIN {X 0,Y 277.327,Z 177.937,A -85,B 0,C 180,E1 -17300.781,E2 -17300.781} C_VEL
LIN {X 0,Y 277.321,Z 177.939,A -85,B 0,C 180,E1 -17304.171,E2 -17304.171} C_VEL
LIN {X 0,Y 277.325,Z 177.943,A -85,B 0,C 180,E1 -17307.505,E2 -17307.505} C_VEL
LIN {X 0,Y 277.274,Z 177.945,A -85,B 0,C 180,E1 -17310.482,E2 -17310.482} C_VEL
LIN {X 0,Y 277.249,Z 177.949,A -85,B 0,C 180,E1 -17313.896,E2 -17313.896} C_VEL
LIN {X 0,Y 277.27,Z 177.949,A -85,B 0,C 180,E1 -17317.47,E2 -17317.47} C_VEL
LIN {X 0,Y 277.292,Z 178.026,A -85,B 0,C 180,E1 -17319.009,E2 -17319.009} C_VEL
LIN {X 0,Y 278.123,Z 182.653,A -85,B 0,C 180,E1 -17323.022,E2 -17323.022} C_VEL
LIN {X 0,Y 279.073,Z 187.763,A -85,B 0,C 180,E1 -17327.16,E2 -17327.16} C_VEL
LIN {X 0,Y 279.99,Z 192.972,A -85,B 0,C 180,E1 -17331.133,E2 -17331.133} C_VEL
LIN {X 0,Y 280.053,Z 196.161,A -85,B 0,C 180,E1 -17333.423,E2 -17333.423} C_VEL
LIN {X 0,Y 279.385,Z 200.551,A -85,B 0,C 180,E1 -17336.399,E2 -17336.399} C_VEL
LIN {X 0,Y 278.259,Z 206.721,A -85,B 0,C 180,E1 -17340.494,E2 -17340.494} C_VEL
LIN {X 0,Y 277.291,Z 213.191,A -85,B 0,C 180,E1 -17344.668,E2 -17344.668} C_VEL
LIN {X 0,Y 279.729,Z 227.233,A -85,B 0,C 180,E1 -17345.557,E2 -17345.557} C_VEL
LIN {X 0,Y 281.438,Z 239.512,A -85,B 0,C 180,E1 -17346.585,E2 -17346.585} C_VEL
LIN {X 0,Y 282.679,Z 252.438,A -85,B 0,C 180,E1 -17347.932,E2 -17347.932} C_VEL
LIN {X 0,Y 283.193,Z 263.117,A -85,B 0,C 180,E1 -17349.29,E2 -17349.29} C_VEL
LIN {X 0,Y 281.425,Z 273.863,A -85,B 0,C 180,E1 -17350.867,E2 -17350.867} C_VEL
LIN {X 0,Y 279.838,Z 284.225,A -85,B 0,C 180,E1 -17352.781,E2 -17352.781} C_VEL
LIN {X 0,Y 278.509,Z 292.339,A -85,B 0,C 180,E1 -17354.636,E2 -17354.636} C_VEL
LIN {X 0,Y 277.273,Z 300.007,A -85,B 0,C 180,E1 -17356.814,E2 -17356.814} C_VEL
LIN {X 0,Y 276.397,Z 306.172,A -85,B 0,C 180,E1 -17359.006,E2 -17359.006} C_VEL
LIN {X 0,Y 275.828,Z 311.055,A -85,B 0,C 180,E1 -17361.206,E2 -17361.206} C_VEL
LIN {X 0,Y 275.526,Z 314.792,A -85,B 0,C 180,E1 -17363.409,E2 -17363.409} C_VEL
LIN {X 0,Y 275.444,Z 317.487,A -85,B 0,C 180,E1 -17365.61,E2 -17365.61} C_VEL
LIN {X 0,Y 275.415,Z 318.737,A -85,B 0,C 180,E1 -17367.075,E2 -17367.075} C_VEL
LIN {X 0,Y 275.413,Z 319.58,A -85,B 0,C 180,E1 -17368.538,E2 -17368.538} C_VEL
LIN {X 0,Y 275.51,Z 319.982,A -85,B 0,C 180,E1 -17370,E2 -17370} C_VEL
LIN {X 0,Y 275.398,Z 319.551,A -85,B 0,C 180,E1 -17372.926,E2 -17372.926} C_VEL
LIN {X 0,Y 275.42,Z 317.745,A -85,B 0,C 180,E1 -17375.623,E2 -17375.623} C_VEL
LIN {X 0,Y 275.681,Z 314.889,A -85,B 0,C 180,E1 -17378.06,E2 -17378.06} C_VEL
LIN {X 0,Y 276.184,Z 311.267,A -85,B 0,C 180,E1 -17380.261,E2 -17380.261} C_VEL
LIN {X 0,Y 276.978,Z 306.569,A -85,B 0,C 180,E1 -17382.456,E2 -17382.456} C_VEL
LIN {X 0,Y 278.515,Z 299.536,A -85,B 0,C 180,E1 -17384.99,E2 -17384.99} C_VEL
LIN {X 0,Y 280.164,Z 292.013,A -85,B 0,C 180,E1 -17387.143,E2 -17387.143} C_VEL
LIN {X 0,Y 282.049,Z 282.75,A -85,B 0,C 180,E1 -17389.279,E2 -17389.279} C_VEL
LIN {X 0,Y 284.315,Z 272.195,A -85,B 0,C 180,E1 -17391.194,E2 -17391.194} C_VEL
LIN {X 0,Y 285.571,Z 265.375,A -85,B 0,C 180,E1 -17392.234,E2 -17392.234} C_VEL
LIN {X 0,Y 285.748,Z 253.341,A -85,B 0,C 180,E1 -17393.922,E2 -17393.922} C_VEL
LIN {X 0,Y 285.189,Z 243.201,A -85,B 0,C 180,E1 -17395.155,E2 -17395.155} C_VEL
LIN {X 0,Y 283.422,Z 231.037,A -85,B 0,C 180,E1 -17396.51,E2 -17396.51} C_VEL
LIN {X 0,Y 280.797,Z 219.651,A -85,B 0,C 180,E1 -17397.662,E2 -17397.662} C_VEL
LIN {X 0,Y 278.276,Z 211.038,A -85,B 0,C 180,E1 -17398.464,E2 -17398.464} C_VEL
LIN {X 0,Y 278.211,Z 210.314,A -85,B 0,C 180,E1 -17398.549,E2 -17398.549} C_VEL
LIN {X 0,Y 279.673,Z 203.148,A -85,B 0,C 180,E1 -17403.563,E2 -17403.563} C_VEL
LIN {X 0,Y 280.442,Z 198.983,A -85,B 0,C 180,E1 -17406.684,E2 -17406.684} C_VEL
LIN {X 0,Y 280.456,Z 196.115,A -85,B 0,C 180,E1 -17409.027,E2 -17409.027} C_VEL
LIN {X 0,Y 279.829,Z 192.063,A -85,B 0,C 180,E1 -17412.697,E2 -17412.697} C_VEL
LIN {X 0,Y 279.015,Z 187.752,A -85,B 0,C 180,E1 -17417.148,E2 -17417.148} C_VEL
LIN {X 0,Y 278.378,Z 184.153,A -85,B 0,C 180,E1 -17421.503,E2 -17421.503} C_VEL
LIN {X 0,Y 278.015,Z 182.069,A -85,B 0,C 180,E1 -17424.449,E2 -17424.449} C_VEL
LIN {X 0,Y 277.614,Z 180.026,A -85,B 0,C 180,E1 -17427.884,E2 -17427.884} C_VEL
LIN {X 0,Y 277.353,Z 178.383,A -85,B 0,C 180,E1 -17431.219,E2 -17431.219} C_VEL
LIN {X 0,Y 277.361,Z 177.933,A -85,B 0,C 180,E1 -17432.864,E2 -17432.864} C_VEL
LIN {X 0,Y 277.333,Z 177.939,A -85,B 0,C 180,E1 -17436.079,E2 -17436.079} C_VEL
LIN {X 0,Y 277.339,Z 177.94,A -85,B 0,C 180,E1 -17440.765,E2 -17440.765} C_VEL
LIN {X 0,Y 277.414,Z 177.93,A -85,B 0,C 180,E1 -17445.324,E2 -17445.324} C_VEL
LIN {X 0,Y 277.511,Z 177.918,A -85,B 0,C 180,E1 -17449.788,E2 -17449.788} C_VEL
LIN {X 0,Y 277.657,Z 177.9,A -85,B 0,C 180,E1 -17452.728,E2 -17452.728} C_VEL
LIN {X 0,Y 277.826,Z 177.88,A -85,B 0,C 180,E1 -17458.55,E2 -17458.55} C_VEL
LIN {X 0,Y 277.986,Z 178.863,A -85,B 0,C 180,E1 -17461.448,E2 -17461.448} C_VEL
LIN {X 0,Y 278.057,Z 181.228,A -85,B 0,C 180,E1 -17466.77,E2 -17466.77} C_VEL
LIN {X 0,Y 278.025,Z 182.711,A -85,B 0,C 180,E1 -17469.647,E2 -17469.647} C_VEL
LIN {X 0,Y 277.722,Z 184.727,A -85,B 0,C 180,E1 -17473.164,E2 -17473.164} C_VEL
LIN {X 0,Y 277.391,Z 186.776,A -85,B 0,C 180,E1 -17476.479,E2 -17476.479} C_VEL
LIN {X 0,Y 278.529,Z 189.88,A -85,B 0,C 180,E1 -17476.844,E2 -17476.844} C_VEL
LIN {X 0,Y 282.776,Z 199.71,A -85,B 0,C 180,E1 -17478.099,E2 -17478.099} C_VEL
LIN {X 0,Y 286.212,Z 209.953,A -85,B 0,C 180,E1 -17479.452,E2 -17479.452} C_VEL
LIN {X 0,Y 288.675,Z 220.132,A -85,B 0,C 180,E1 -17480.857,E2 -17480.857} C_VEL
LIN {X 0,Y 289.59,Z 225.583,A -85,B 0,C 180,E1 -17481.655,E2 -17481.655} C_VEL
LIN {X 0,Y 287.564,Z 237.468,A -85,B 0,C 180,E1 -17483.208,E2 -17483.208} C_VEL
LIN {X 0,Y 285.574,Z 247.747,A -85,B 0,C 180,E1 -17484.925,E2 -17484.925} C_VEL
LIN {X 0,Y 283.512,Z 256.951,A -85,B 0,C 180,E1 -17486.822,E2 -17486.822} C_VEL
LIN {X 0,Y 281.831,Z 264.155,A -85,B 0,C 180,E1 -17488.664,E2 -17488.664} C_VEL
LIN {X 0,Y 280.188,Z 270.572,A -85,B 0,C 180,E1 -17490.683,E2 -17490.683} C_VEL
LIN {X 0,Y 278.815,Z 275.772,A -85,B 0,C 180,E1 -17492.726,E2 -17492.726} C_VEL
LIN {X 0,Y 277.818,Z 279.727,A -85,B 0,C 180,E1 -17494.692,E2 -17494.692} C_VEL
LIN {X 0,Y 277.011,Z 282.726,A -85,B 0,C 180,E1 -17496.628,E2 -17496.628} C_VEL
LIN {X 0,Y 276.52,Z 284.412,A -85,B 0,C 180,E1 -17498.01,E2 -17498.01} C_VEL
LIN {X 0,Y 275.918,Z 286.245,A -85,B 0,C 180,E1 -17500.169,E2 -17500.169} C_VEL
LIN {X 0,Y 275.577,Z 287.171,A -85,B 0,C 180,E1 -17502.303,E2 -17502.303} C_VEL
LIN {X 0,Y 275.395,Z 287.257,A -85,B 0,C 180,E1 -17504.393,E2 -17504.393} C_VEL
LIN {X 0,Y 275.355,Z 286.559,A -85,B 0,C 180,E1 -17506.438,E2 -17506.438} C_VEL
LIN {X 0,Y 275.534,Z 285.083,A -85,B 0,C 180,E1 -17508.457,E2 -17508.457} C_VEL
LIN {X 0,Y 275.904,Z 282.817,A -85,B 0,C 180,E1 -17510.445,E2 -17510.445} C_VEL
LIN {X 0,Y 276.336,Z 279.832,A -85,B 0,C 180,E1 -17512.382,E2 -17512.382} C_VEL
LIN {X 0,Y 277.047,Z 274.963,A -85,B 0,C 180,E1 -17514.777,E2 -17514.777} C_VEL
LIN {X 0,Y 277.921,Z 269.248,A -85,B 0,C 180,E1 -17516.957,E2 -17516.957} C_VEL
LIN {X 0,Y 278.923,Z 262.773,A -85,B 0,C 180,E1 -17518.946,E2 -17518.946} C_VEL
LIN {X 0,Y 280.306,Z 254.568,A -85,B 0,C 180,E1 -17520.982,E2 -17520.982} C_VEL
LIN {X 0,Y 281.752,Z 244.887,A -85,B 0,C 180,E1 -17522.92,E2 -17522.92} C_VEL
LIN {X 0,Y 283.228,Z 234.118,A -85,B 0,C 180,E1 -17524.656,E2 -17524.656} C_VEL
LIN {X 0,Y 284.696,Z 222.317,A -85,B 0,C 180,E1 -17526.148,E2 -17526.148} C_VEL
LIN {X 0,Y 285.083,Z 218.556,A -85,B 0,C 180,E1 -17526.557,E2 -17526.557} C_VEL
LIN {X 0,Y 282.704,Z 206.39,A -85,B 0,C 180,E1 -17527.915,E2 -17527.915} C_VEL
LIN {X 0,Y 279.447,Z 193.699,A -85,B 0,C 180,E1 -17529.095,E2 -17529.095} C_VEL
LIN {X 0,Y 276.352,Z 182.9,A -85,B 0,C 180,E1 -17529.909,E2 -17529.909} C_VEL
LIN {X 0,Y 276.572,Z 179.717,A -85,B 0,C 180,E1 -17533.768,E2 -17533.768} C_VEL
LIN {X 0,Y 276.738,Z 178.489,A -85,B 0,C 180,E1 -17535.288,E2 -17535.288} C_VEL
LIN {X 0,Y 276.829,Z 178.002,A -85,B 0,C 180,E1 -17536.792,E2 -17536.792} C_VEL
LIN {X 0,Y 277.516,Z 177.914,A -85,B 0,C 180,E1 -17541.26,E2 -17541.26} C_VEL
LIN {X 0,Y 277.558,Z 177.914,A -85,B 0,C 180,E1 -17544.187,E2 -17544.187} C_VEL
LIN {X 0,Y 277.819,Z 177.878,A -85,B 0,C 180,E1 -17548.55,E2 -17548.55} C_VEL
LIN {X 0,Y 277.819,Z 177.876,A -85,B 0,C 180,E1 -17551.449,E2 -17551.449} C_VEL
LIN {X 0,Y 277.65,Z 177.899,A -85,B 0,C 180,E1 -17557.271,E2 -17557.271} C_VEL
LIN {X 0,Y 277.503,Z 177.916,A -85,B 0,C 180,E1 -17560.211,E2 -17560.211} C_VEL
LIN {X 0,Y 277.431,Z 177.926,A -85,B 0,C 180,E1 -17564.674,E2 -17564.674} C_VEL
LIN {X 0,Y 277.342,Z 177.937,A -85,B 0,C 180,E1 -17569.234,E2 -17569.234} C_VEL
LIN {X 0,Y 277.325,Z 177.94,A -85,B 0,C 180,E1 -17573.921,E2 -17573.921} C_VEL
LIN {X 0,Y 277.319,Z 177.941,A -85,B 0,C 180,E1 -17577.504,E2 -17577.504} C_VEL
LIN {X 0,Y 277.269,Z 177.945,A -85,B 0,C 180,E1 -17580.482,E2 -17580.482} C_VEL
LIN {X 0,Y 277.243,Z 177.947,A -85,B 0,C 180,E1 -17583.896,E2 -17583.896} C_VEL
LIN {X 0,Y 277.262,Z 177.946,A -85,B 0,C 180,E1 -17587.47,E2 -17587.47} C_VEL
LIN {X 0,Y 277.207,Z 177.956,A -85,B 0,C 180,E1 -17591.237,E2 -17591.237} C_VEL
LIN {X 0,Y 277.213,Z 177.953,A -85,B 0,C 180,E1 -17595.224,E2 -17595.224} C_VEL
LIN {X 0,Y 277.22,Z 177.949,A -85,B 0,C 180,E1 -17599.513,E2 -17599.513} C_VEL
LIN {X 0,Y 277.263,Z 177.946,A -85,B 0,C 180,E1 -17602.531,E2 -17602.531} C_VEL
LIN {X 0,Y 277.245,Z 177.948,A -85,B 0,C 180,E1 -17606.105,E2 -17606.105} C_VEL
LIN {X 0,Y 277.26,Z 177.942,A -85,B 0,C 180,E1 -17609.539,E2 -17609.539} C_VEL
LIN {X 0,Y 277.354,Z 177.934,A -85,B 0,C 180,E1 -17612.865,E2 -17612.865} C_VEL
LIN {X 0,Y 277.327,Z 177.938,A -85,B 0,C 180,E1 -17616.08,E2 -17616.08} C_VEL
LIN {X 0,Y 277.345,Z 177.936,A -85,B 0,C 180,E1 -17620.767,E2 -17620.767} C_VEL
LIN {X 0,Y 277.435,Z 177.919,A -85,B 0,C 180,E1 -17625.327,E2 -17625.327} C_VEL
LIN {X 0,Y 277.461,Z 177.922,A -85,B 0,C 180,E1 -17629.788,E2 -17629.788} C_VEL
LIN {X 0,Y 277.641,Z 177.899,A -85,B 0,C 180,E1 -17632.73,E2 -17632.73} C_VEL
LIN {X 0,Y 277.822,Z 177.874,A -85,B 0,C 180,E1 -17638.551,E2 -17638.551} C_VEL
LIN {X 0,Y 277.821,Z 177.876,A -85,B 0,C 180,E1 -17641.45,E2 -17641.45} C_VEL
LIN {X 0,Y 277.612,Z 177.901,A -85,B 0,C 180,E1 -17647.273,E2 -17647.273} C_VEL
LIN {X 0,Y 277.459,Z 177.922,A -85,B 0,C 180,E1 -17650.214,E2 -17650.214} C_VEL
LIN {X 0,Y 277.406,Z 177.927,A -85,B 0,C 180,E1 -17652.194,E2 -17652.194} C_VEL
LIN {X 0,Y 276.716,Z 178.016,A -85,B 0,C 180,E1 -17653.407,E2 -17653.407} C_VEL
LIN {X 0,Y 273.842,Z 178.374,A -85,B 0,C 180,E1 -17655.382,E2 -17655.382} C_VEL
LIN {X 0,Y 271.41,Z 178.675,A -85,B 0,C 180,E1 -17656.987,E2 -17656.987} C_VEL
LIN {X 0,Y 270.362,Z 178.804,A -85,B 0,C 180,E1 -17658.231,E2 -17658.231} C_VEL
LIN {X 0,Y 270.274,Z 178.813,A -85,B 0,C 180,E1 -17658.652,E2 -17658.652} C_VEL
LIN {X 0,Y 270.246,Z 178.822,A -85,B 0,C 180,E1 -17661.352,E2 -17661.352} C_VEL
LIN {X 0,Y 270.276,Z 178.816,A -85,B 0,C 180,E1 -17664.586,E2 -17664.586} C_VEL
LIN {X 0,Y 270.271,Z 178.819,A -85,B 0,C 180,E1 -17667.909,E2 -17667.909} C_VEL
LIN {X 0,Y 270.186,Z 178.832,A -85,B 0,C 180,E1 -17671.349,E2 -17671.349} C_VEL
LIN {X 0,Y 270.204,Z 178.828,A -85,B 0,C 180,E1 -17674.906,E2 -17674.906} C_VEL
LIN {X 0,Y 270.263,Z 178.941,A -85,B 0,C 180,E1 -17678.617,E2 -17678.617} C_VEL
LIN {X 0,Y 271.006,Z 183.175,A -85,B 0,C 180,E1 -17682.398,E2 -17682.398} C_VEL
LIN {X 0,Y 271.876,Z 187.918,A -85,B 0,C 180,E1 -17686.37,E2 -17686.37} C_VEL
LIN {X 0,Y 272.699,Z 192.354,A -85,B 0,C 180,E1 -17689.887,E2 -17689.887} C_VEL
LIN {X 0,Y 273.074,Z 196.395,A -85,B 0,C 180,E1 -17692.925,E2 -17692.925} C_VEL
LIN {X 0,Y 272.308,Z 201.327,A -85,B 0,C 180,E1 -17696.379,E2 -17696.379} C_VEL
LIN {X 0,Y 271.181,Z 207.382,A -85,B 0,C 180,E1 -17700.501,E2 -17700.501} C_VEL
LIN {X 0,Y 270.346,Z 213.04,A -85,B 0,C 180,E1 -17704.119,E2 -17704.119} C_VEL
LIN {X 0,Y 272.691,Z 226.382,A -85,B 0,C 180,E1 -17704.99,E2 -17704.99} C_VEL
LIN {X 0,Y 274.261,Z 237.868,A -85,B 0,C 180,E1 -17705.962,E2 -17705.962} C_VEL
LIN {X 0,Y 275.526,Z 249.976,A -85,B 0,C 180,E1 -17707.236,E2 -17707.236} C_VEL
LIN {X 0,Y 276.221,Z 261.754,A -85,B 0,C 180,E1 -17708.742,E2 -17708.742} C_VEL
LIN {X 0,Y 275.85,Z 265.717,A -85,B 0,C 180,E1 -17709.299,E2 -17709.299} C_VEL
LIN {X 0,Y 274.175,Z 275.956,A -85,B 0,C 180,E1 -17710.924,E2 -17710.924} C_VEL
LIN {X 0,Y 272.589,Z 285.915,A -85,B 0,C 180,E1 -17712.917,E2 -17712.917} C_VEL
LIN {X 0,Y 271.146,Z 294.215,A -85,B 0,C 180,E1 -17714.978,E2 -17714.978} C_VEL
LIN {X 0,Y 269.947,Z 301.468,A -85,B 0,C 180,E1 -17717.215,E2 -17717.215} C_VEL
LIN {X 0,Y 269.188,Z 307.271,A -85,B 0,C 180,E1 -17719.47,E2 -17719.47} C_VEL
LIN {X 0,Y 268.656,Z 311.815,A -85,B 0,C 180,E1 -17721.728,E2 -17721.728} C_VEL
LIN {X 0,Y 268.42,Z 315.558,A -85,B 0,C 180,E1 -17724.244,E2 -17724.244} C_VEL
LIN {X 0,Y 268.345,Z 318.225,A -85,B 0,C 180,E1 -17726.998,E2 -17726.998} C_VEL
LIN {X 0,Y 268.333,Z 319.093,A -85,B 0,C 180,E1 -17728.499,E2 -17728.499} C_VEL
LIN {X 0,Y 268.423,Z 319.542,A -85,B 0,C 180,E1 -17730,E2 -17730} C_VEL
LIN {X 0,Y 268.325,Z 319.159,A -85,B 0,C 180,E1 -17733.003,E2 -17733.003} C_VEL
LIN {X 0,Y 268.339,Z 317.555,A -85,B 0,C 180,E1 -17735.581,E2 -17735.581} C_VEL
LIN {X 0,Y 268.612,Z 314.602,A -85,B 0,C 180,E1 -17738.274,E2 -17738.274} C_VEL
LIN {X 0,Y 269.167,Z 311.022,A -85,B 0,C 180,E1 -17740.532,E2 -17740.532} C_VEL
LIN {X 0,Y 270.019,Z 306.397,A -85,B 0,C 180,E1 -17742.782,E2 -17742.782} C_VEL
LIN {X 0,Y 271.651,Z 299.481,A -85,B 0,C 180,E1 -17745.378,E2 -17745.378} C_VEL
LIN {X 0,Y 273.383,Z 292.05,A -85,B 0,C 180,E1 -17747.582,E2 -17747.582} C_VEL
LIN {X 0,Y 275.356,Z 282.926,A -85,B 0,C 180,E1 -17749.767,E2 -17749.767} C_VEL
LIN {X 0,Y 277.737,Z 272.501,A -85,B 0,C 180,E1 -17751.721,E2 -17751.721} C_VEL
LIN {X 0,Y 278.958,Z 265.813,A -85,B 0,C 180,E1 -17752.79,E2 -17752.79} C_VEL
LIN {X 0,Y 279.26,Z 254.331,A -85,B 0,C 180,E1 -17754.482,E2 -17754.482} C_VEL
LIN {X 0,Y 278.797,Z 244.19,A -85,B 0,C 180,E1 -17755.795,E2 -17755.795} C_VEL
LIN {X 0,Y 277.212,Z 232.661,A -85,B 0,C 180,E1 -17757.152,E2 -17757.152} C_VEL
LIN {X 0,Y 274.477,Z 220.436,A -85,B 0,C 180,E1 -17758.477,E2 -17758.477} C_VEL
LIN {X 0,Y 271.51,Z 210.547,A -85,B 0,C 180,E1 -17759.493,E2 -17759.493} C_VEL
LIN {X 0,Y 271.41,Z 209.796,A -85,B 0,C 180,E1 -17759.579,E2 -17759.579} C_VEL
LIN {X 0,Y 272.67,Z 204.175,A -85,B 0,C 180,E1 -17763.643,E2 -17763.643} C_VEL
LIN {X 0,Y 273.333,Z 200.769,A -85,B 0,C 180,E1 -17766.256,E2 -17766.256} C_VEL
LIN {X 0,Y 273.564,Z 198.538,A -85,B 0,C 180,E1 -17768.067,E2 -17768.067} C_VEL
LIN {X 0,Y 273.004,Z 194.199,A -85,B 0,C 180,E1 -17772.015,E2 -17772.015} C_VEL
LIN {X 0,Y 272.189,Z 190.071,A -85,B 0,C 180,E1 -17776.301,E2 -17776.301} C_VEL
LIN {X 0,Y 271.561,Z 186.208,A -85,B 0,C 180,E1 -17780.933,E2 -17780.933} C_VEL
LIN {X 0,Y 271.225,Z 184.406,A -85,B 0,C 180,E1 -17783.444,E2 -17783.444} C_VEL
LIN {X 0,Y 270.813,Z 182.237,A -85,B 0,C 180,E1 -17786.976,E2 -17786.976} C_VEL
LIN {X 0,Y 270.527,Z 180.483,A -85,B 0,C 180,E1 -17790.422,E2 -17790.422} C_VEL
LIN {X 0,Y 270.32,Z 179.163,A -85,B 0,C 180,E1 -17793.769,E2 -17793.769} C_VEL
LIN {X 0,Y 270.281,Z 178.814,A -85,B 0,C 180,E1 -17795.519,E2 -17795.519} C_VEL
LIN {X 0,Y 270.301,Z 178.813,A -85,B 0,C 180,E1 -17800.244,E2 -17800.244} C_VEL
LIN {X 0,Y 270.381,Z 178.805,A -85,B 0,C 180,E1 -17804.933,E2 -17804.933} C_VEL
LIN {X 0,Y 270.446,Z 178.798,A -85,B 0,C 180,E1 -17809.518,E2 -17809.518} C_VEL
LIN {X 0,Y 270.616,Z 178.778,A -85,B 0,C 180,E1 -17812.538,E2 -17812.538} C_VEL
LIN {X 0,Y 270.661,Z 178.908,A -85,B 0,C 180,E1 -17817.022,E2 -17817.022} C_VEL
LIN {X 0,Y 271.031,Z 179.794,A -85,B 0,C 180,E1 -17819.999,E2 -17819.999} C_VEL
LIN {X 0,Y 270.981,Z 180.945,A -85,B 0,C 180,E1 -17822.973,E2 -17822.973} C_VEL
LIN {X 0,Y 271.133,Z 182.921,A -85,B 0,C 180,E1 -17827.446,E2 -17827.446} C_VEL
LIN {X 0,Y 270.957,Z 184.481,A -85,B 0,C 180,E1 -17830.46,E2 -17830.46} C_VEL
LIN {X 0,Y 270.668,Z 186.193,A -85,B 0,C 180,E1 -17833.513,E2 -17833.513} C_VEL
LIN {X 0,Y 270.496,Z 187.42,A -85,B 0,C 180,E1 -17835.453,E2 -17835.453} C_VEL
LIN {X 0,Y 271.661,Z 190.493,A -85,B 0,C 180,E1 -17835.82,E2 -17835.82} C_VEL
LIN {X 0,Y 276.273,Z 200.858,A -85,B 0,C 180,E1 -17837.269,E2 -17837.269} C_VEL
LIN {X 0,Y 279.857,Z 211.646,A -85,B 0,C 180,E1 -17838.768,E2 -17838.768} C_VEL
LIN {X 0,Y 282.251,Z 221.571,A -85,B 0,C 180,E1 -17840.234,E2 -17840.234} C_VEL
LIN {X 0,Y 283.172,Z 227.138,A -85,B 0,C 180,E1 -17841.092,E2 -17841.092} C_VEL
LIN {X 0,Y 281.13,Z 238.541,A -85,B 0,C 180,E1 -17842.645,E2 -17842.645} C_VEL
LIN {X 0,Y 279.038,Z 248.788,A -85,B 0,C 180,E1 -17844.41,E2 -17844.41} C_VEL
LIN {X 0,Y 276.952,Z 257.491,A -85,B 0,C 180,E1 -17846.257,E2 -17846.257} C_VEL
LIN {X 0,Y 275.135,Z 264.855,A -85,B 0,C 180,E1 -17848.2,E2 -17848.2} C_VEL
LIN {X 0,Y 273.166,Z 271.994,A -85,B 0,C 180,E1 -17850.56,E2 -17850.56} C_VEL
LIN {X 0,Y 271.624,Z 277.536,A -85,B 0,C 180,E1 -17852.911,E2 -17852.911} C_VEL
LIN {X 0,Y 270.39,Z 282.139,A -85,B 0,C 180,E1 -17855.525,E2 -17855.525} C_VEL
LIN {X 0,Y 269.851,Z 283.843,A -85,B 0,C 180,E1 -17856.798,E2 -17856.798} C_VEL
LIN {X 0,Y 269.178,Z 285.883,A -85,B 0,C 180,E1 -17858.8,E2 -17858.8} C_VEL
LIN {X 0,Y 268.709,Z 287.174,A -85,B 0,C 180,E1 -17860.833,E2 -17860.833} C_VEL
LIN {X 0,Y 268.446,Z 287.743,A -85,B 0,C 180,E1 -17862.896,E2 -17862.896} C_VEL
LIN {X 0,Y 268.273,Z 287.557,A -85,B 0,C 180,E1 -17865.016,E2 -17865.016} C_VEL
LIN {X 0,Y 268.332,Z 286.514,A -85,B 0,C 180,E1 -17867.168,E2 -17867.168} C_VEL
LIN {X 0,Y 268.6,Z 284.583,A -85,B 0,C 180,E1 -17869.357,E2 -17869.357} C_VEL
LIN {X 0,Y 269.056,Z 281.669,A -85,B 0,C 180,E1 -17871.593,E2 -17871.593} C_VEL
LIN {X 0,Y 269.642,Z 277.586,A -85,B 0,C 180,E1 -17873.899,E2 -17873.899} C_VEL
LIN {X 0,Y 270.499,Z 272.178,A -85,B 0,C 180,E1 -17876.242,E2 -17876.242} C_VEL
LIN {X 0,Y 271.642,Z 265.12,A -85,B 0,C 180,E1 -17878.624,E2 -17878.624} C_VEL
LIN {X 0,Y 273.18,Z 256.149,A -85,B 0,C 180,E1 -17881.008,E2 -17881.008} C_VEL
LIN {X 0,Y 274.692,Z 246.503,A -85,B 0,C 180,E1 -17883.04,E2 -17883.04} C_VEL
LIN {X 0,Y 276.315,Z 235.147,A -85,B 0,C 180,E1 -17884.948,E2 -17884.948} C_VEL
LIN {X 0,Y 277.811,Z 223.803,A -85,B 0,C 180,E1 -17886.442,E2 -17886.442} C_VEL
LIN {X 0,Y 278.126,Z 218.966,A -85,B 0,C 180,E1 -17886.999,E2 -17886.999} C_VEL
LIN {X 0,Y 275.796,Z 207.156,A -85,B 0,C 180,E1 -17888.364,E2 -17888.364} C_VEL
LIN {X 0,Y 272.522,Z 194.291,A -85,B 0,C 180,E1 -17889.607,E2 -17889.607} C_VEL
LIN {X 0,Y 269.377,Z 183.292,A -85,B 0,C 180,E1 -17890.471,E2 -17890.471} C_VEL
LIN {X 0,Y 269.65,Z 179.723,A -85,B 0,C 180,E1 -17894.892,E2 -17894.892} C_VEL
LIN {X 0,Y 269.742,Z 178.887,A -85,B 0,C 180,E1 -17896.438,E2 -17896.438} C_VEL
LIN {X 0,Y 270.456,Z 178.794,A -85,B 0,C 180,E1 -17901.03,E2 -17901.03} C_VEL
LIN {X 0,Y 270.527,Z 178.789,A -85,B 0,C 180,E1 -17904.035,E2 -17904.035} C_VEL
LIN {X 0,Y 270.784,Z 178.755,A -85,B 0,C 180,E1 -17908.513,E2 -17908.513} C_VEL
LIN {X 0,Y 270.785,Z 178.753,A -85,B 0,C 180,E1 -17911.487,E2 -17911.487} C_VEL
LIN {X 0,Y 270.608,Z 178.777,A -85,B 0,C 180,E1 -17917.461,E2 -17917.461} C_VEL
LIN {X 0,Y 270.438,Z 178.795,A -85,B 0,C 180,E1 -17920.481,E2 -17920.481} C_VEL
LIN {X 0,Y 270.4,Z 178.803,A -85,B 0,C 180,E1 -17925.065,E2 -17925.065} C_VEL
LIN {X 0,Y 270.299,Z 178.818,A -85,B 0,C 180,E1 -17929.756,E2 -17929.756} C_VEL
LIN {X 0,Y 270.27,Z 178.817,A -85,B 0,C 180,E1 -17934.586,E2 -17934.586} C_VEL
LIN {X 0,Y 270.266,Z 178.818,A -85,B 0,C 180,E1 -17937.909,E2 -17937.909} C_VEL
LIN {X 0,Y 270.181,Z 178.833,A -85,B 0,C 180,E1 -17941.348,E2 -17941.348} C_VEL
LIN {X 0,Y 270.198,Z 178.826,A -85,B 0,C 180,E1 -17944.906,E2 -17944.906} C_VEL
LIN {X 0,Y 270.194,Z 178.825,A -85,B 0,C 180,E1 -17948.711,E2 -17948.711} C_VEL
LIN {X 0,Y 270.169,Z 178.832,A -85,B 0,C 180,E1 -17953.251,E2 -17953.251} C_VEL
LIN {X 0,Y 270.172,Z 178.824,A -85,B 0,C 180,E1 -17957.443,E2 -17957.443} C_VEL
LIN {X 0,Y 270.204,Z 178.825,A -85,B 0,C 180,E1 -17961.375,E2 -17961.375} C_VEL
LIN {X 0,Y 270.199,Z 178.827,A -85,B 0,C 180,E1 -17965.095,E2 -17965.095} C_VEL
LIN {X 0,Y 270.198,Z 178.823,A -85,B 0,C 180,E1 -17969.131,E2 -17969.131} C_VEL
LIN {X 0,Y 270.261,Z 178.813,A -85,B 0,C 180,E1 -17972.147,E2 -17972.147} C_VEL
LIN {X 0,Y 270.276,Z 178.815,A -85,B 0,C 180,E1 -17975.52,E2 -17975.52} C_VEL
LIN {X 0,Y 270.301,Z 178.815,A -85,B 0,C 180,E1 -17980.245,E2 -17980.245} C_VEL
LIN {X 0,Y 270.403,Z 178.796,A -85,B 0,C 180,E1 -17984.936,E2 -17984.936} C_VEL
LIN {X 0,Y 270.413,Z 178.798,A -85,B 0,C 180,E1 -17989.519,E2 -17989.519} C_VEL
LIN {X 0,Y 270.599,Z 178.777,A -85,B 0,C 180,E1 -17992.539,E2 -17992.539} C_VEL
LIN {X 0,Y 270.788,Z 178.75,A -85,B 0,C 180,E1 -17998.514,E2 -17998.514} C_VEL
LIN {X 0,Y 270.787,Z 178.752,A -85,B 0,C 180,E1 -18001.488,E2 -18001.488} C_VEL
LIN {X 0,Y 270.572,Z 178.779,A -85,B 0,C 180,E1 -18007.463,E2 -18007.463} C_VEL
LIN {X 0,Y 270.411,Z 178.798,A -85,B 0,C 180,E1 -18010.483,E2 -18010.483} C_VEL
LIN {X 0,Y 270.405,Z 178.8,A -85,B 0,C 180,E1 -18015.065,E2 -18015.065} C_VEL
LIN {X 0,Y 270.274,Z 178.813,A -85,B 0,C 180,E1 -18018.652,E2 -18018.652} C_VEL
LIN {X 0,Y 269.6,Z 178.902,A -85,B 0,C 180,E1 -18019.895,E2 -18019.895} C_VEL
LIN {X 0,Y 266.754,Z 179.257,A -85,B 0,C 180,E1 -18021.919,E2 -18021.919} C_VEL
LIN {X 0,Y 264.339,Z 179.56,A -85,B 0,C 180,E1 -18023.565,E2 -18023.565} C_VEL
LIN {X 0,Y 263.298,Z 179.687,A -85,B 0,C 180,E1 -18024.84,E2 -18024.84} C_VEL
LIN {X 0,Y 263.21,Z 179.699,A -85,B 0,C 180,E1 -18025.273,E2 -18025.273} C_VEL
LIN {X 0,Y 263.167,Z 179.703,A -85,B 0,C 180,E1 -18028.732,E2 -18028.732} C_VEL
LIN {X 0,Y 263.135,Z 179.706,A -85,B 0,C 180,E1 -18032.289,E2 -18032.289} C_VEL
LIN {X 0,Y 263.185,Z 179.702,A -85,B 0,C 180,E1 -18036.764,E2 -18036.764} C_VEL
LIN {X 0,Y 263.202,Z 179.78,A -85,B 0,C 180,E1 -18038.13,E2 -18038.13} C_VEL
LIN {X 0,Y 263.895,Z 183.733,A -85,B 0,C 180,E1 -18041.782,E2 -18041.782} C_VEL
LIN {X 0,Y 264.743,Z 188.37,A -85,B 0,C 180,E1 -18045.788,E2 -18045.788} C_VEL
LIN {X 0,Y 265.718,Z 193.618,A -85,B 0,C 180,E1 -18050.088,E2 -18050.088} C_VEL
LIN {X 0,Y 266.035,Z 196.858,A -85,B 0,C 180,E1 -18052.584,E2 -18052.584} C_VEL
LIN {X 0,Y 265.617,Z 200.332,A -85,B 0,C 180,E1 -18055.109,E2 -18055.109} C_VEL
LIN {X 0,Y 264.305,Z 206.783,A -85,B 0,C 180,E1 -18059.654,E2 -18059.654} C_VEL
LIN {X 0,Y 263.387,Z 212.428,A -85,B 0,C 180,E1 -18063.533,E2 -18063.533} C_VEL
LIN {X 0,Y 265.778,Z 226.45,A -85,B 0,C 180,E1 -18064.473,E2 -18064.473} C_VEL
LIN {X 0,Y 267.482,Z 238.95,A -85,B 0,C 180,E1 -18065.585,E2 -18065.585} C_VEL
LIN {X 0,Y 268.663,Z 250.809,A -85,B 0,C 180,E1 -18066.897,E2 -18066.897} C_VEL
LIN {X 0,Y 269.253,Z 261.822,A -85,B 0,C 180,E1 -18068.365,E2 -18068.365} C_VEL
LIN {X 0,Y 268.968,Z 265.758,A -85,B 0,C 180,E1 -18068.944,E2 -18068.944} C_VEL
LIN {X 0,Y 267.249,Z 275.91,A -85,B 0,C 180,E1 -18070.61,E2 -18070.61} C_VEL
LIN {X 0,Y 265.578,Z 285.898,A -85,B 0,C 180,E1 -18072.678,E2 -18072.678} C_VEL
LIN {X 0,Y 264.047,Z 294.721,A -85,B 0,C 180,E1 -18074.959,E2 -18074.959} C_VEL
LIN {X 0,Y 262.81,Z 301.767,A -85,B 0,C 180,E1 -18077.255,E2 -18077.255} C_VEL
LIN {X 0,Y 261.965,Z 308.217,A -85,B 0,C 180,E1 -18079.958,E2 -18079.958} C_VEL
LIN {X 0,Y 261.493,Z 312.441,A -85,B 0,C 180,E1 -18082.277,E2 -18082.277} C_VEL
LIN {X 0,Y 261.347,Z 315.198,A -85,B 0,C 180,E1 -18084.265,E2 -18084.265} C_VEL
LIN {X 0,Y 261.277,Z 317.712,A -85,B 0,C 180,E1 -18086.916,E2 -18086.916} C_VEL
LIN {X 0,Y 261.256,Z 318.605,A -85,B 0,C 180,E1 -18088.459,E2 -18088.459} C_VEL
LIN {X 0,Y 261.338,Z 319.096,A -85,B 0,C 180,E1 -18090,E2 -18090} C_VEL
LIN {X 0,Y 261.246,Z 319.13,A -85,B 0,C 180,E1 -18091.542,E2 -18091.542} C_VEL
LIN {X 0,Y 261.253,Z 318.766,A -85,B 0,C 180,E1 -18093.084,E2 -18093.084} C_VEL
LIN {X 0,Y 261.298,Z 316.858,A -85,B 0,C 180,E1 -18096.176,E2 -18096.176} C_VEL
LIN {X 0,Y 261.563,Z 314.319,A -85,B 0,C 180,E1 -18098.499,E2 -18098.499} C_VEL
LIN {X 0,Y 262.141,Z 310.807,A -85,B 0,C 180,E1 -18100.817,E2 -18100.817} C_VEL
LIN {X 0,Y 263.079,Z 306.246,A -85,B 0,C 180,E1 -18103.125,E2 -18103.125} C_VEL
LIN {X 0,Y 264.799,Z 299.438,A -85,B 0,C 180,E1 -18105.786,E2 -18105.786} C_VEL
LIN {X 0,Y 266.618,Z 292.087,A -85,B 0,C 180,E1 -18108.043,E2 -18108.043} C_VEL
LIN {X 0,Y 268.677,Z 283.079,A -85,B 0,C 180,E1 -18110.279,E2 -18110.279} C_VEL
LIN {X 0,Y 270.92,Z 273.928,A -85,B 0,C 180,E1 -18112.096,E2 -18112.096} C_VEL
LIN {X 0,Y 272.307,Z 267.448,A -85,B 0,C 180,E1 -18113.178,E2 -18113.178} C_VEL
LIN {X 0,Y 272.798,Z 255.404,A -85,B 0,C 180,E1 -18115.07,E2 -18115.07} C_VEL
LIN {X 0,Y 272.423,Z 245.158,A -85,B 0,C 180,E1 -18116.467,E2 -18116.467} C_VEL
LIN {X 0,Y 270.732,Z 232.534,A -85,B 0,C 180,E1 -18118.039,E2 -18118.039} C_VEL
LIN {X 0,Y 267.728,Z 219.618,A -85,B 0,C 180,E1 -18119.542,E2 -18119.542} C_VEL
LIN {X 0,Y 265.378,Z 212.309,A -85,B 0,C 180,E1 -18120.375,E2 -18120.375} C_VEL
LIN {X 0,Y 264.643,Z 209.253,A -85,B 0,C 180,E1 -18120.69,E2 -18120.69} C_VEL
LIN {X 0,Y 265.663,Z 205.176,A -85,B 0,C 180,E1 -18123.749,E2 -18123.749} C_VEL
LIN {X 0,Y 266.361,Z 201.804,A -85,B 0,C 180,E1 -18126.418,E2 -18126.418} C_VEL
LIN {X 0,Y 266.561,Z 200.232,A -85,B 0,C 180,E1 -18127.723,E2 -18127.723} C_VEL
LIN {X 0,Y 266.317,Z 197.636,A -85,B 0,C 180,E1 -18130.066,E2 -18130.066} C_VEL
LIN {X 0,Y 265.739,Z 194.214,A -85,B 0,C 180,E1 -18133.443,E2 -18133.443} C_VEL
LIN {X 0,Y 265.243,Z 191.45,A -85,B 0,C 180,E1 -18136.455,E2 -18136.455} C_VEL
LIN {X 0,Y 264.696,Z 188.222,A -85,B 0,C 180,E1 -18140.414,E2 -18140.414} C_VEL
LIN {X 0,Y 264.198,Z 185.618,A -85,B 0,C 180,E1 -18144.18,E2 -18144.18} C_VEL
LIN {X 0,Y 263.785,Z 183.131,A -85,B 0,C 180,E1 -18148.494,E2 -18148.494} C_VEL
LIN {X 0,Y 263.472,Z 181.182,A -85,B 0,C 180,E1 -18153.033,E2 -18153.033} C_VEL
LIN {X 0,Y 263.26,Z 180.139,A -85,B 0,C 180,E1 -18156.393,E2 -18156.393} C_VEL
LIN {X 0,Y 263.266,Z 179.687,A -85,B 0,C 180,E1 -18159.693,E2 -18159.693} C_VEL
LIN {X 0,Y 263.327,Z 179.684,A -85,B 0,C 180,E1 -18164.52,E2 -18164.52} C_VEL
LIN {X 0,Y 263.378,Z 179.679,A -85,B 0,C 180,E1 -18169.234,E2 -18169.234} C_VEL
LIN {X 0,Y 263.577,Z 179.654,A -85,B 0,C 180,E1 -18172.338,E2 -18172.338} C_VEL
LIN {X 0,Y 263.709,Z 180.446,A -85,B 0,C 180,E1 -18176.944,E2 -18176.944} C_VEL
LIN {X 0,Y 264.099,Z 181.3,A -85,B 0,C 180,E1 -18179.999,E2 -18179.999} C_VEL
LIN {X 0,Y 264.036,Z 182.445,A -85,B 0,C 180,E1 -18183.051,E2 -18183.051} C_VEL
LIN {X 0,Y 264.116,Z 184.005,A -85,B 0,C 180,E1 -18186.789,E2 -18186.789} C_VEL
LIN {X 0,Y 264.054,Z 185.562,A -85,B 0,C 180,E1 -18190.006,E2 -18190.006} C_VEL
LIN {X 0,Y 263.589,Z 187.917,A -85,B 0,C 180,E1 -18194.277,E2 -18194.277} C_VEL
LIN {X 0,Y 264.744,Z 191.023,A -85,B 0,C 180,E1 -18194.705,E2 -18194.705} C_VEL
LIN {X 0,Y 268.908,Z 199.939,A -85,B 0,C 180,E1 -18196.044,E2 -18196.044} C_VEL
LIN {X 0,Y 272.514,Z 209.741,A -85,B 0,C 180,E1 -18197.515,E2 -18197.515} C_VEL
LIN {X 0,Y 275.402,Z 220.567,A -85,B 0,C 180,E1 -18199.18,E2 -18199.18} C_VEL
LIN {X 0,Y 276.794,Z 229.451,A -85,B 0,C 180,E1 -18200.608,E2 -18200.608} C_VEL
LIN {X 0,Y 274.608,Z 240.28,A -85,B 0,C 180,E1 -18202.157,E2 -18202.157} C_VEL
LIN {X 0,Y 272.387,Z 250.384,A -85,B 0,C 180,E1 -18203.976,E2 -18203.976} C_VEL
LIN {X 0,Y 270.201,Z 258.995,A -85,B 0,C 180,E1 -18205.904,E2 -18205.904} C_VEL
LIN {X 0,Y 268.07,Z 267.014,A -85,B 0,C 180,E1 -18208.157,E2 -18208.157} C_VEL
LIN {X 0,Y 266.076,Z 273.766,A -85,B 0,C 180,E1 -18210.55,E2 -18210.55} C_VEL
LIN {X 0,Y 264.489,Z 279.062,A -85,B 0,C 180,E1 -18213.005,E2 -18213.005} C_VEL
LIN {X 0,Y 263.498,Z 282.513,A -85,B 0,C 180,E1 -18215.09,E2 -18215.09} C_VEL
LIN {X 0,Y 262.343,Z 285.918,A -85,B 0,C 180,E1 -18218.035,E2 -18218.035} C_VEL
LIN {X 0,Y 261.571,Z 287.886,A -85,B 0,C 180,E1 -18221.208,E2 -18221.208} C_VEL
LIN {X 0,Y 261.228,Z 288.094,A -85,B 0,C 180,E1 -18224.385,E2 -18224.385} C_VEL
LIN {X 0,Y 261.197,Z 287.249,A -85,B 0,C 180,E1 -18226.591,E2 -18226.591} C_VEL
LIN {X 0,Y 261.435,Z 285.547,A -85,B 0,C 180,E1 -18228.824,E2 -18228.824} C_VEL
LIN {X 0,Y 261.864,Z 282.887,A -85,B 0,C 180,E1 -18231.105,E2 -18231.105} C_VEL
LIN {X 0,Y 262.567,Z 278.195,A -85,B 0,C 180,E1 -18233.923,E2 -18233.923} C_VEL
LIN {X 0,Y 263.454,Z 272.689,A -85,B 0,C 180,E1 -18236.39,E2 -18236.39} C_VEL
LIN {X 0,Y 264.568,Z 266.206,A -85,B 0,C 180,E1 -18238.666,E2 -18238.666} C_VEL
LIN {X 0,Y 265.833,Z 258.861,A -85,B 0,C 180,E1 -18240.742,E2 -18240.742} C_VEL
LIN {X 0,Y 267.433,Z 249.329,A -85,B 0,C 180,E1 -18242.916,E2 -18242.916} C_VEL
LIN {X 0,Y 268.884,Z 239.902,A -85,B 0,C 180,E1 -18244.659,E2 -18244.659} C_VEL
LIN {X 0,Y 270.443,Z 229.196,A -85,B 0,C 180,E1 -18246.246,E2 -18246.246} C_VEL
LIN {X 0,Y 271.339,Z 220.416,A -85,B 0,C 180,E1 -18247.334,E2 -18247.334} C_VEL
LIN {X 0,Y 269.144,Z 209.026,A -85,B 0,C 180,E1 -18248.715,E2 -18248.715} C_VEL
LIN {X 0,Y 265.938,Z 196.304,A -85,B 0,C 180,E1 -18250.007,E2 -18250.007} C_VEL
LIN {X 0,Y 262.368,Z 183.692,A -85,B 0,C 180,E1 -18251.047,E2 -18251.047} C_VEL
LIN {X 0,Y 262.552,Z 180.962,A -85,B 0,C 180,E1 -18254.501,E2 -18254.501} C_VEL
LIN {X 0,Y 262.635,Z 179.772,A -85,B 0,C 180,E1 -18256.064,E2 -18256.064} C_VEL
LIN {X 0,Y 263.356,Z 179.679,A -85,B 0,C 180,E1 -18260.887,E2 -18260.887} C_VEL
LIN {X 0,Y 263.497,Z 179.664,A -85,B 0,C 180,E1 -18263.875,E2 -18263.875} C_VEL
LIN {X 0,Y 263.749,Z 179.631,A -85,B 0,C 180,E1 -18268.473,E2 -18268.473} C_VEL
LIN {X 0,Y 263.749,Z 179.629,A -85,B 0,C 180,E1 -18271.527,E2 -18271.527} C_VEL
LIN {X 0,Y 263.569,Z 179.655,A -85,B 0,C 180,E1 -18277.661,E2 -18277.661} C_VEL
LIN {X 0,Y 263.371,Z 179.675,A -85,B 0,C 180,E1 -18280.766,E2 -18280.766} C_VEL
LIN {X 0,Y 263.348,Z 179.684,A -85,B 0,C 180,E1 -18285.478,E2 -18285.478} C_VEL
LIN {X 0,Y 263.265,Z 179.691,A -85,B 0,C 180,E1 -18290.306,E2 -18290.306} C_VEL
LIN {X 0,Y 263.204,Z 179.7,A -85,B 0,C 180,E1 -18295.292,E2 -18295.292} C_VEL
LIN {X 0,Y 263.162,Z 179.702,A -85,B 0,C 180,E1 -18298.731,E2 -18298.731} C_VEL
LIN {X 0,Y 263.129,Z 179.707,A -85,B 0,C 180,E1 -18302.289,E2 -18302.289} C_VEL
LIN {X 0,Y 263.178,Z 179.696,A -85,B 0,C 180,E1 -18306.763,E2 -18306.763} C_VEL
LIN {X 0,Y 263.122,Z 179.708,A -85,B 0,C 180,E1 -18311.594,E2 -18311.594} C_VEL
LIN {X 0,Y 263.125,Z 179.704,A -85,B 0,C 180,E1 -18316.018,E2 -18316.018} C_VEL
LIN {X 0,Y 263.103,Z 179.706,A -85,B 0,C 180,E1 -18320.128,E2 -18320.128} C_VEL
LIN {X 0,Y 263.16,Z 179.702,A -85,B 0,C 180,E1 -18324.019,E2 -18324.019} C_VEL
LIN {X 0,Y 263.131,Z 179.704,A -85,B 0,C 180,E1 -18327.712,E2 -18327.712} C_VEL
LIN {X 0,Y 263.194,Z 179.691,A -85,B 0,C 180,E1 -18331.786,E2 -18331.786} C_VEL
LIN {X 0,Y 263.225,Z 179.694,A -85,B 0,C 180,E1 -18335.201,E2 -18335.201} C_VEL
LIN {X 0,Y 263.268,Z 179.688,A -85,B 0,C 180,E1 -18339.695,E2 -18339.695} C_VEL
LIN {X 0,Y 263.351,Z 179.675,A -85,B 0,C 180,E1 -18344.523,E2 -18344.523} C_VEL
LIN {X 0,Y 263.355,Z 179.677,A -85,B 0,C 180,E1 -18349.234,E2 -18349.234} C_VEL
LIN {X 0,Y 263.558,Z 179.656,A -85,B 0,C 180,E1 -18352.339,E2 -18352.339} C_VEL
LIN {X 0,Y 263.752,Z 179.627,A -85,B 0,C 180,E1 -18358.474,E2 -18358.474} C_VEL
LIN {X 0,Y 263.751,Z 179.629,A -85,B 0,C 180,E1 -18361.528,E2 -18361.528} C_VEL
LIN {X 0,Y 263.534,Z 179.656,A -85,B 0,C 180,E1 -18367.663,E2 -18367.663} C_VEL
LIN {X 0,Y 263.354,Z 179.676,A -85,B 0,C 180,E1 -18370.767,E2 -18370.767} C_VEL
LIN {X 0,Y 263.353,Z 179.681,A -85,B 0,C 180,E1 -18375.479,E2 -18375.479} C_VEL
LIN {X 0,Y 263.27,Z 179.689,A -85,B 0,C 180,E1 -18380.307,E2 -18380.307} C_VEL
LIN {X 0,Y 263.21,Z 179.699,A -85,B 0,C 180,E1 -18385.273,E2 -18385.273} C_VEL
LIN {X 0,Y 262.532,Z 179.791,A -85,B 0,C 180,E1 -18386.55,E2 -18386.55} C_VEL
LIN {X 0,Y 259.67,Z 180.15,A -85,B 0,C 180,E1 -18388.631,E2 -18388.631} C_VEL
LIN {X 0,Y 257.229,Z 180.449,A -85,B 0,C 180,E1 -18390.324,E2 -18390.324} C_VEL
LIN {X 0,Y 256.162,Z 180.577,A -85,B 0,C 180,E1 -18391.637,E2 -18391.637} C_VEL
LIN {X 0,Y 256.063,Z 180.587,A -85,B 0,C 180,E1 -18392.082,E2 -18392.082} C_VEL
LIN {X 0,Y 256.084,Z 180.588,A -85,B 0,C 180,E1 -18395.193,E2 -18395.193} C_VEL
LIN {X 0,Y 256.16,Z 180.595,A -85,B 0,C 180,E1 -18397.633,E2 -18397.633} C_VEL
LIN {X 0,Y 257.036,Z 185.688,A -85,B 0,C 180,E1 -18402.418,E2 -18402.418} C_VEL
LIN {X 0,Y 258.009,Z 191,A -85,B 0,C 180,E1 -18407.08,E2 -18407.08} C_VEL
LIN {X 0,Y 258.781,Z 195.093,A -85,B 0,C 180,E1 -18410.478,E2 -18410.478} C_VEL
LIN {X 0,Y 258.88,Z 198.773,A -85,B 0,C 180,E1 -18413.327,E2 -18413.327} C_VEL
LIN {X 0,Y 258.224,Z 202.497,A -85,B 0,C 180,E1 -18416.087,E2 -18416.087} C_VEL
LIN {X 0,Y 257.005,Z 208.648,A -85,B 0,C 180,E1 -18420.513,E2 -18420.513} C_VEL
LIN {X 0,Y 256.412,Z 212.063,A -85,B 0,C 180,E1 -18422.926,E2 -18422.926} C_VEL
LIN {X 0,Y 258.812,Z 225.989,A -85,B 0,C 180,E1 -18423.903,E2 -18423.903} C_VEL
LIN {X 0,Y 260.62,Z 239.382,A -85,B 0,C 180,E1 -18425.142,E2 -18425.142} C_VEL
LIN {X 0,Y 261.733,Z 250.791,A -85,B 0,C 180,E1 -18426.448,E2 -18426.448} C_VEL
LIN {X 0,Y 262.293,Z 261.845,A -85,B 0,C 180,E1 -18427.968,E2 -18427.968} C_VEL
LIN {X 0,Y 262.096,Z 265.775,A -85,B 0,C 180,E1 -18428.571,E2 -18428.571} C_VEL
LIN {X 0,Y 260.333,Z 275.833,A -85,B 0,C 180,E1 -18430.278,E2 -18430.278} C_VEL
LIN {X 0,Y 258.643,Z 285.403,A -85,B 0,C 180,E1 -18432.315,E2 -18432.315} C_VEL
LIN {X 0,Y 257.119,Z 293.85,A -85,B 0,C 180,E1 -18434.544,E2 -18434.544} C_VEL
LIN {X 0,Y 255.851,Z 301.009,A -85,B 0,C 180,E1 -18436.902,E2 -18436.902} C_VEL
LIN {X 0,Y 254.922,Z 307.527,A -85,B 0,C 180,E1 -18439.677,E2 -18439.677} C_VEL
LIN {X 0,Y 254.423,Z 311.812,A -85,B 0,C 180,E1 -18442.061,E2 -18442.061} C_VEL
LIN {X 0,Y 254.254,Z 314.879,A -85,B 0,C 180,E1 -18444.332,E2 -18444.332} C_VEL
LIN {X 0,Y 254.211,Z 317.194,A -85,B 0,C 180,E1 -18446.831,E2 -18446.831} C_VEL
LIN {X 0,Y 254.181,Z 318.112,A -85,B 0,C 180,E1 -18448.416,E2 -18448.416} C_VEL
LIN {X 0,Y 254.255,Z 318.634,A -85,B 0,C 180,E1 -18450,E2 -18450} C_VEL
LIN {X 0,Y 254.171,Z 318.715,A -85,B 0,C 180,E1 -18451.585,E2 -18451.585} C_VEL
LIN {X 0,Y 254.16,Z 318.378,A -85,B 0,C 180,E1 -18453.171,E2 -18453.171} C_VEL
LIN {X 0,Y 254.233,Z 316.529,A -85,B 0,C 180,E1 -18456.349,E2 -18456.349} C_VEL
LIN {X 0,Y 254.376,Z 314.989,A -85,B 0,C 180,E1 -18457.941,E2 -18457.941} C_VEL
LIN {X 0,Y 254.875,Z 311.877,A -85,B 0,C 180,E1 -18460.325,E2 -18460.325} C_VEL
LIN {X 0,Y 255.721,Z 307.74,A -85,B 0,C 180,E1 -18462.701,E2 -18462.701} C_VEL
LIN {X 0,Y 257.367,Z 301.476,A -85,B 0,C 180,E1 -18465.441,E2 -18465.441} C_VEL
LIN {X 0,Y 259.126,Z 294.78,A -85,B 0,C 180,E1 -18467.755,E2 -18467.755} C_VEL
LIN {X 0,Y 261.263,Z 286.494,A -85,B 0,C 180,E1 -18470.058,E2 -18470.058} C_VEL
LIN {X 0,Y 263.381,Z 278.138,A -85,B 0,C 180,E1 -18471.937,E2 -18471.937} C_VEL
LIN {X 0,Y 265.65,Z 269.107,A -85,B 0,C 180,E1 -18473.588,E2 -18473.588} C_VEL
LIN {X 0,Y 266.33,Z 257.444,A -85,B 0,C 180,E1 -18475.522,E2 -18475.522} C_VEL
LIN {X 0,Y 266.22,Z 247.996,A -85,B 0,C 180,E1 -18476.909,E2 -18476.909} C_VEL
LIN {X 0,Y 264.887,Z 236.054,A -85,B 0,C 180,E1 -18478.528,E2 -18478.528} C_VEL
LIN {X 0,Y 262.405,Z 223.8,A -85,B 0,C 180,E1 -18480.064,E2 -18480.064} C_VEL
LIN {X 0,Y 259.062,Z 212.602,A -85,B 0,C 180,E1 -18481.444,E2 -18481.444} C_VEL
LIN {X 0,Y 258.043,Z 209.621,A -85,B 0,C 180,E1 -18481.799,E2 -18481.799} C_VEL
LIN {X 0,Y 257.952,Z 208.707,A -85,B 0,C 180,E1 -18481.9,E2 -18481.9} C_VEL
LIN {X 0,Y 259.147,Z 204.077,A -85,B 0,C 180,E1 -18485.55,E2 -18485.55} C_VEL
LIN {X 0,Y 259.528,Z 200.925,A -85,B 0,C 180,E1 -18488.249,E2 -18488.249} C_VEL
LIN {X 0,Y 259.11,Z 197.388,A -85,B 0,C 180,E1 -18491.646,E2 -18491.646} C_VEL
LIN {X 0,Y 258.515,Z 194.227,A -85,B 0,C 180,E1 -18495.021,E2 -18495.021} C_VEL
LIN {X 0,Y 257.917,Z 190.78,A -85,B 0,C 180,E1 -18499.157,E2 -18499.157} C_VEL
LIN {X 0,Y 257.442,Z 187.967,A -85,B 0,C 180,E1 -18503.087,E2 -18503.087} C_VEL
LIN {X 0,Y 257.027,Z 185.726,A -85,B 0,C 180,E1 -18506.847,E2 -18506.847} C_VEL
LIN {X 0,Y 256.683,Z 183.631,A -85,B 0,C 180,E1 -18511.184,E2 -18511.184} C_VEL
LIN {X 0,Y 256.505,Z 182.351,A -85,B 0,C 180,E1 -18514.712,E2 -18514.712} C_VEL
LIN {X 0,Y 256.298,Z 181.281,A -85,B 0,C 180,E1 -18519.115,E2 -18519.115} C_VEL
LIN {X 0,Y 256.272,Z 180.714,A -85,B 0,C 180,E1 -18523.709,E2 -18523.709} C_VEL
LIN {X 0,Y 256.294,Z 180.671,A -85,B 0,C 180,E1 -18527.327,E2 -18527.327} C_VEL
LIN {X 0,Y 256.54,Z 180.863,A -85,B 0,C 180,E1 -18530.538,E2 -18530.538} C_VEL
LIN {X 0,Y 256.626,Z 181.33,A -85,B 0,C 180,E1 -18533.71,E2 -18533.71} C_VEL
LIN {X 0,Y 257.008,Z 182.379,A -85,B 0,C 180,E1 -18538.432,E2 -18538.432} C_VEL
LIN {X 0,Y 257.159,Z 183.357,A -85,B 0,C 180,E1 -18541.565,E2 -18541.565} C_VEL
LIN {X 0,Y 257.159,Z 185.414,A -85,B 0,C 180,E1 -18546.781,E2 -18546.781} C_VEL
LIN {X 0,Y 257.061,Z 187.001,A -85,B 0,C 180,E1 -18550.185,E2 -18550.185} C_VEL
LIN {X 0,Y 256.718,Z 188.517,A -85,B 0,C 180,E1 -18553.052,E2 -18553.052} C_VEL
LIN {X 0,Y 257.752,Z 191.407,A -85,B 0,C 180,E1 -18553.45,E2 -18553.45} C_VEL
LIN {X 0,Y 259.128,Z 193.916,A -85,B 0,C 180,E1 -18553.877,E2 -18553.877} C_VEL
LIN {X 0,Y 263.482,Z 203.641,A -85,B 0,C 180,E1 -18555.469,E2 -18555.469} C_VEL
LIN {X 0,Y 267.214,Z 214.483,A -85,B 0,C 180,E1 -18557.21,E2 -18557.21} C_VEL
LIN {X 0,Y 269.675,Z 225.326,A -85,B 0,C 180,E1 -18559.011,E2 -18559.011} C_VEL
LIN {X 0,Y 270.455,Z 230.604,A -85,B 0,C 180,E1 -18559.921,E2 -18559.921} C_VEL
LIN {X 0,Y 268.297,Z 241.289,A -85,B 0,C 180,E1 -18561.513,E2 -18561.513} C_VEL
LIN {X 0,Y 265.987,Z 251.174,A -85,B 0,C 180,E1 -18563.348,E2 -18563.348} C_VEL
LIN {X 0,Y 263.758,Z 259.379,A -85,B 0,C 180,E1 -18565.234,E2 -18565.234} C_VEL
LIN {X 0,Y 261.519,Z 267.331,A -85,B 0,C 180,E1 -18567.521,E2 -18567.521} C_VEL
LIN {X 0,Y 259.457,Z 273.96,A -85,B 0,C 180,E1 -18569.911,E2 -18569.911} C_VEL
LIN {X 0,Y 257.817,Z 279.145,A -85,B 0,C 180,E1 -18572.322,E2 -18572.322} C_VEL
LIN {X 0,Y 256.402,Z 283.587,A -85,B 0,C 180,E1 -18575.141,E2 -18575.141} C_VEL
LIN {X 0,Y 255.532,Z 285.97,A -85,B 0,C 180,E1 -18577.233,E2 -18577.233} C_VEL
LIN {X 0,Y 254.855,Z 287.643,A -85,B 0,C 180,E1 -18579.453,E2 -18579.453} C_VEL
LIN {X 0,Y 254.404,Z 288.525,A -85,B 0,C 180,E1 -18581.764,E2 -18581.764} C_VEL
LIN {X 0,Y 254.176,Z 288.568,A -85,B 0,C 180,E1 -18584.035,E2 -18584.035} C_VEL
LIN {X 0,Y 254.116,Z 287.825,A -85,B 0,C 180,E1 -18586.257,E2 -18586.257} C_VEL
LIN {X 0,Y 254.297,Z 286.314,A -85,B 0,C 180,E1 -18588.448,E2 -18588.448} C_VEL
LIN {X 0,Y 254.884,Z 282.587,A -85,B 0,C 180,E1 -18591.654,E2 -18591.654} C_VEL
LIN {X 0,Y 255.46,Z 278.914,A -85,B 0,C 180,E1 -18593.875,E2 -18593.875} C_VEL
LIN {X 0,Y 256.276,Z 274.175,A -85,B 0,C 180,E1 -18596.115,E2 -18596.115} C_VEL
LIN {X 0,Y 257.475,Z 267.07,A -85,B 0,C 180,E1 -18598.76,E2 -18598.76} C_VEL
LIN {X 0,Y 259.015,Z 258.597,A -85,B 0,C 180,E1 -18601.208,E2 -18601.208} C_VEL
LIN {X 0,Y 260.555,Z 249.635,A -85,B 0,C 180,E1 -18603.289,E2 -18603.289} C_VEL
LIN {X 0,Y 262.092,Z 239.986,A -85,B 0,C 180,E1 -18605.11,E2 -18605.11} C_VEL
LIN {X 0,Y 263.819,Z 228.256,A -85,B 0,C 180,E1 -18606.863,E2 -18606.863} C_VEL
LIN {X 0,Y 264.533,Z 222.798,A -85,B 0,C 180,E1 -18607.548,E2 -18607.548} C_VEL
LIN {X 0,Y 263.18,Z 214.187,A -85,B 0,C 180,E1 -18608.663,E2 -18608.663} C_VEL
LIN {X 0,Y 260.29,Z 201.785,A -85,B 0,C 180,E1 -18610.069,E2 -18610.069} C_VEL
LIN {X 0,Y 256.629,Z 188.689,A -85,B 0,C 180,E1 -18611.281,E2 -18611.281} C_VEL
LIN {X 0,Y 255.297,Z 184.103,A -85,B 0,C 180,E1 -18611.647,E2 -18611.647} C_VEL
LIN {X 0,Y 255.577,Z 180.992,A -85,B 0,C 180,E1 -18615.671,E2 -18615.671} C_VEL
LIN {X 0,Y 255.959,Z 180.6,A -85,B 0,C 180,E1 -18618.918,E2 -18618.918} C_VEL
LIN {X 0,Y 256.442,Z 180.544,A -85,B 0,C 180,E1 -18622.124,E2 -18622.124} C_VEL
LIN {X 0,Y 256.331,Z 180.555,A -85,B 0,C 180,E1 -18625.282,E2 -18625.282} C_VEL
LIN {X 0,Y 256.712,Z 180.508,A -85,B 0,C 180,E1 -18628.431,E2 -18628.431} C_VEL
LIN {X 0,Y 256.712,Z 180.506,A -85,B 0,C 180,E1 -18631.569,E2 -18631.569} C_VEL
LIN {X 0,Y 256.537,Z 180.533,A -85,B 0,C 180,E1 -18637.873,E2 -18637.873} C_VEL
LIN {X 0,Y 256.307,Z 180.555,A -85,B 0,C 180,E1 -18641.066,E2 -18641.066} C_VEL
LIN {X 0,Y 256.297,Z 180.561,A -85,B 0,C 180,E1 -18645.915,E2 -18645.915} C_VEL
LIN {X 0,Y 256.215,Z 180.57,A -85,B 0,C 180,E1 -18650.891,E2 -18650.891} C_VEL
LIN {X 0,Y 256.185,Z 180.574,A -85,B 0,C 180,E1 -18655.139,E2 -18655.139} C_VEL
LIN {X 0,Y 256.1,Z 180.585,A -85,B 0,C 180,E1 -18659.601,E2 -18659.601} C_VEL
LIN {X 0,Y 256.064,Z 180.589,A -85,B 0,C 180,E1 -18663.293,E2 -18663.293} C_VEL
LIN {X 0,Y 256.111,Z 180.579,A -85,B 0,C 180,E1 -18667.271,E2 -18667.271} C_VEL
LIN {X 0,Y 256.052,Z 180.592,A -85,B 0,C 180,E1 -18671.204,E2 -18671.204} C_VEL
LIN {X 0,Y 256.059,Z 180.585,A -85,B 0,C 180,E1 -18675.53,E2 -18675.53} C_VEL
LIN {X 0,Y 256.052,Z 180.583,A -85,B 0,C 180,E1 -18678.797,E2 -18678.797} C_VEL
LIN {X 0,Y 256.128,Z 180.581,A -85,B 0,C 180,E1 -18682.868,E2 -18682.868} C_VEL
LIN {X 0,Y 256.066,Z 180.589,A -85,B 0,C 180,E1 -18686.708,E2 -18686.708} C_VEL
LIN {X 0,Y 256.102,Z 180.578,A -85,B 0,C 180,E1 -18690.4,E2 -18690.4} C_VEL
LIN {X 0,Y 256.187,Z 180.572,A -85,B 0,C 180,E1 -18694.862,E2 -18694.862} C_VEL
LIN {X 0,Y 256.217,Z 180.567,A -85,B 0,C 180,E1 -18699.11,E2 -18699.11} C_VEL
LIN {X 0,Y 256.3,Z 180.553,A -85,B 0,C 180,E1 -18704.086,E2 -18704.086} C_VEL
LIN {X 0,Y 256.298,Z 180.557,A -85,B 0,C 180,E1 -18708.934,E2 -18708.934} C_VEL
LIN {X 0,Y 256.515,Z 180.534,A -85,B 0,C 180,E1 -18712.127,E2 -18712.127} C_VEL
LIN {X 0,Y 256.501,Z 180.525,A -85,B 0,C 180,E1 -18716.859,E2 -18716.859} C_VEL
LIN {X 0,Y 256.766,Z 180.499,A -85,B 0,C 180,E1 -18720.001,E2 -18720.001} C_VEL
LIN {X 0,Y 256.497,Z 180.533,A -85,B 0,C 180,E1 -18723.142,E2 -18723.142} C_VEL
LIN {X 0,Y 256.496,Z 180.531,A -85,B 0,C 180,E1 -18727.875,E2 -18727.875} C_VEL
LIN {X 0,Y 256.295,Z 180.558,A -85,B 0,C 180,E1 -18732.673,E2 -18732.673} C_VEL
LIN {X 0,Y 256.285,Z 180.558,A -85,B 0,C 180,E1 -18736.303,E2 -18736.303} C_VEL
LIN {X 0,Y 256.187,Z 180.572,A -85,B 0,C 180,E1 -18741.137,E2 -18741.137} C_VEL
LIN {X 0,Y 256.181,Z 180.574,A -85,B 0,C 180,E1 -18745.244,E2 -18745.244} C_VEL
LIN {X 0,Y 256.105,Z 180.585,A -85,B 0,C 180,E1 -18749.602,E2 -18749.602} C_VEL
LIN {X 0,Y 256.063,Z 180.587,A -85,B 0,C 180,E1 -18752.082,E2 -18752.082} C_VEL
LIN {X 0,Y 255.365,Z 180.679,A -85,B 0,C 180,E1 -18753.395,E2 -18753.395} C_VEL
LIN {X 0,Y 252.547,Z 181.075,A -85,B 0,C 180,E1 -18755.538,E2 -18755.538} C_VEL
LIN {X 0,Y 250.266,Z 181.908,A -85,B 0,C 180,E1 -18757.269,E2 -18757.269} C_VEL
LIN {X 0,Y 249.404,Z 182.927,A -85,B 0,C 180,E1 -18758.596,E2 -18758.596} C_VEL
LIN {X 0,Y 249.394,Z 183.356,A -85,B 0,C 180,E1 -18759.04,E2 -18759.04} C_VEL
LIN {X 0,Y 250.196,Z 187.602,A -85,B 0,C 180,E1 -18763.085,E2 -18763.085} C_VEL
LIN {X 0,Y 251.158,Z 192.906,A -85,B 0,C 180,E1 -18767.811,E2 -18767.811} C_VEL
LIN {X 0,Y 251.885,Z 197.16,A -85,B 0,C 180,E1 -18771.376,E2 -18771.376} C_VEL
LIN {X 0,Y 251.672,Z 200.621,A -85,B 0,C 180,E1 -18774.096,E2 -18774.096} C_VEL
LIN {X 0,Y 250.647,Z 205.544,A -85,B 0,C 180,E1 -18777.809,E2 -18777.809} C_VEL
LIN {X 0,Y 249.483,Z 211.786,A -85,B 0,C 180,E1 -18782.303,E2 -18782.303} C_VEL
LIN {X 0,Y 251.857,Z 225.571,A -85,B 0,C 180,E1 -18783.303,E2 -18783.303} C_VEL
LIN {X 0,Y 253.604,Z 238.073,A -85,B 0,C 180,E1 -18784.495,E2 -18784.495} C_VEL
LIN {X 0,Y 254.835,Z 251.315,A -85,B 0,C 180,E1 -18786.055,E2 -18786.055} C_VEL
LIN {X 0,Y 255.377,Z 263.051,A -85,B 0,C 180,E1 -18787.766,E2 -18787.766} C_VEL
LIN {X 0,Y 254.796,Z 268.029,A -85,B 0,C 180,E1 -18788.564,E2 -18788.564} C_VEL
LIN {X 0,Y 252.897,Z 278.558,A -85,B 0,C 180,E1 -18790.52,E2 -18790.52} C_VEL
LIN {X 0,Y 251.384,Z 287.161,A -85,B 0,C 180,E1 -18792.51,E2 -18792.51} C_VEL
LIN {X 0,Y 249.792,Z 295.508,A -85,B 0,C 180,E1 -18794.915,E2 -18794.915} C_VEL
LIN {X 0,Y 248.517,Z 302.228,A -85,B 0,C 180,E1 -18797.34,E2 -18797.34} C_VEL
LIN {X 0,Y 247.693,Z 308.4,A -85,B 0,C 180,E1 -18800.198,E2 -18800.198} C_VEL
LIN {X 0,Y 247.274,Z 312.38,A -85,B 0,C 180,E1 -18802.652,E2 -18802.652} C_VEL
LIN {X 0,Y 247.129,Z 315.294,A -85,B 0,C 180,E1 -18805.106,E2 -18805.106} C_VEL
LIN {X 0,Y 247.145,Z 316.664,A -85,B 0,C 180,E1 -18806.74,E2 -18806.74} C_VEL
LIN {X 0,Y 247.108,Z 317.611,A -85,B 0,C 180,E1 -18808.371,E2 -18808.371} C_VEL
LIN {X 0,Y 247.175,Z 318.161,A -85,B 0,C 180,E1 -18810,E2 -18810} C_VEL
LIN {X 0,Y 247.097,Z 318.295,A -85,B 0,C 180,E1 -18811.63,E2 -18811.63} C_VEL
LIN {X 0,Y 247.069,Z 317.991,A -85,B 0,C 180,E1 -18813.262,E2 -18813.262} C_VEL
LIN {X 0,Y 247.165,Z 316.197,A -85,B 0,C 180,E1 -18816.531,E2 -18816.531} C_VEL
LIN {X 0,Y 247.311,Z 314.706,A -85,B 0,C 180,E1 -18818.169,E2 -18818.169} C_VEL
LIN {X 0,Y 247.856,Z 311.647,A -85,B 0,C 180,E1 -18820.621,E2 -18820.621} C_VEL
LIN {X 0,Y 248.759,Z 307.589,A -85,B 0,C 180,E1 -18823.063,E2 -18823.063} C_VEL
LIN {X 0,Y 250.518,Z 301.46,A -85,B 0,C 180,E1 -18825.874,E2 -18825.874} C_VEL
LIN {X 0,Y 252.341,Z 294.971,A -85,B 0,C 180,E1 -18828.21,E2 -18828.21} C_VEL
LIN {X 0,Y 254.594,Z 286.672,A -85,B 0,C 180,E1 -18830.607,E2 -18830.607} C_VEL
LIN {X 0,Y 256.806,Z 278.437,A -85,B 0,C 180,E1 -18832.529,E2 -18832.529} C_VEL
LIN {X 0,Y 259.137,Z 269.596,A -85,B 0,C 180,E1 -18834.218,E2 -18834.218} C_VEL
LIN {X 0,Y 259.962,Z 258.472,A -85,B 0,C 180,E1 -18836.173,E2 -18836.173} C_VEL
LIN {X 0,Y 259.928,Z 249.122,A -85,B 0,C 180,E1 -18837.628,E2 -18837.628} C_VEL
LIN {X 0,Y 258.771,Z 237.707,A -85,B 0,C 180,E1 -18839.266,E2 -18839.266} C_VEL
LIN {X 0,Y 256.68,Z 226.373,A -85,B 0,C 180,E1 -18840.805,E2 -18840.805} C_VEL
LIN {X 0,Y 253.495,Z 215.417,A -85,B 0,C 180,E1 -18842.279,E2 -18842.279} C_VEL
LIN {X 0,Y 252.093,Z 211.323,A -85,B 0,C 180,E1 -18842.822,E2 -18842.822} C_VEL
LIN {X 0,Y 251.363,Z 208.112,A -85,B 0,C 180,E1 -18843.224,E2 -18843.224} C_VEL
LIN {X 0,Y 252.255,Z 204.634,A -85,B 0,C 180,E1 -18846.102,E2 -18846.102} C_VEL
LIN {X 0,Y 252.501,Z 201.641,A -85,B 0,C 180,E1 -18848.799,E2 -18848.799} C_VEL
LIN {X 0,Y 252.092,Z 198.445,A -85,B 0,C 180,E1 -18851.997,E2 -18851.997} C_VEL
LIN {X 0,Y 251.327,Z 194.349,A -85,B 0,C 180,E1 -18856.64,E2 -18856.64} C_VEL
LIN {X 0,Y 250.899,Z 191.816,A -85,B 0,C 180,E1 -18859.889,E2 -18859.889} C_VEL
LIN {X 0,Y 250.426,Z 189.118,A -85,B 0,C 180,E1 -18863.888,E2 -18863.888} C_VEL
LIN {X 0,Y 250.062,Z 186.968,A -85,B 0,C 180,E1 -18867.723,E2 -18867.723} C_VEL
LIN {X 0,Y 249.782,Z 185.279,A -85,B 0,C 180,E1 -18871.423,E2 -18871.423} C_VEL
LIN {X 0,Y 249.61,Z 184.019,A -85,B 0,C 180,E1 -18875.017,E2 -18875.017} C_VEL
LIN {X 0,Y 249.391,Z 182.839,A -85,B 0,C 180,E1 -18880.234,E2 -18880.234} C_VEL
LIN {X 0,Y 249.388,Z 182.45,A -85,B 0,C 180,E1 -18883.631,E2 -18883.631} C_VEL
LIN {X 0,Y 249.424,Z 182.428,A -85,B 0,C 180,E1 -18888.624,E2 -18888.624} C_VEL
LIN {X 0,Y 249.679,Z 182.683,A -85,B 0,C 180,E1 -18891.908,E2 -18891.908} C_VEL
LIN {X 0,Y 249.86,Z 183.567,A -85,B 0,C 180,E1 -18896.774,E2 -18896.774} C_VEL
LIN {X 0,Y 250.24,Z 184.356,A -85,B 0,C 180,E1 -18899.999,E2 -18899.999} C_VEL
LIN {X 0,Y 250.149,Z 185.453,A -85,B 0,C 180,E1 -18903.22,E2 -18903.22} C_VEL
LIN {X 0,Y 250.207,Z 186.821,A -85,B 0,C 180,E1 -18906.761,E2 -18906.761} C_VEL
LIN {X 0,Y 250.069,Z 188.453,A -85,B 0,C 180,E1 -18910.373,E2 -18910.373} C_VEL
LIN {X 0,Y 249.899,Z 189.246,A -85,B 0,C 180,E1 -18911.712,E2 -18911.712} C_VEL
LIN {X 0,Y 251.052,Z 192.225,A -85,B 0,C 180,E1 -18912.165,E2 -18912.165} C_VEL
LIN {X 0,Y 252.289,Z 194.338,A -85,B 0,C 180,E1 -18912.576,E2 -18912.576} C_VEL
LIN {X 0,Y 257.102,Z 204.863,A -85,B 0,C 180,E1 -18914.433,E2 -18914.433} C_VEL
LIN {X 0,Y 260.389,Z 214.189,A -85,B 0,C 180,E1 -18916.06,E2 -18916.06} C_VEL
LIN {X 0,Y 263.016,Z 224.73,A -85,B 0,C 180,E1 -18917.895,E2 -18917.895} C_VEL
LIN {X 0,Y 264.13,Z 233.185,A -85,B 0,C 180,E1 -18919.426,E2 -18919.426} C_VEL
LIN {X 0,Y 261.685,Z 243.565,A -85,B 0,C 180,E1 -18921.05,E2 -18921.05} C_VEL
LIN {X 0,Y 259.109,Z 253.702,A -85,B 0,C 180,E1 -18923.067,E2 -18923.067} C_VEL
LIN {X 0,Y 256.557,Z 262.691,A -85,B 0,C 180,E1 -18925.312,E2 -18925.312} C_VEL
LIN {X 0,Y 254.165,Z 270.373,A -85,B 0,C 180,E1 -18927.767,E2 -18927.767} C_VEL
LIN {X 0,Y 252.13,Z 276.403,A -85,B 0,C 180,E1 -18930.218,E2 -18930.218} C_VEL
LIN {X 0,Y 250.505,Z 281.092,A -85,B 0,C 180,E1 -18932.683,E2 -18932.683} C_VEL
LIN {X 0,Y 249.308,Z 284.612,A -85,B 0,C 180,E1 -18935.163,E2 -18935.163} C_VEL
LIN {X 0,Y 248.317,Z 287.028,A -85,B 0,C 180,E1 -18937.582,E2 -18937.582} C_VEL
LIN {X 0,Y 247.482,Z 288.804,A -85,B 0,C 180,E1 -18940.779,E2 -18940.779} C_VEL
LIN {X 0,Y 247.173,Z 289.106,A -85,B 0,C 180,E1 -18943.031,E2 -18943.031} C_VEL
LIN {X 0,Y 247.022,Z 288.616,A -85,B 0,C 180,E1 -18945.337,E2 -18945.337} C_VEL
LIN {X 0,Y 247.116,Z 287.301,A -85,B 0,C 180,E1 -18947.683,E2 -18947.683} C_VEL
LIN {X 0,Y 247.453,Z 285.083,A -85,B 0,C 180,E1 -18950.069,E2 -18950.069} C_VEL
LIN {X 0,Y 248.012,Z 281.834,A -85,B 0,C 180,E1 -18952.507,E2 -18952.507} C_VEL
LIN {X 0,Y 248.75,Z 277.35,A -85,B 0,C 180,E1 -18955.018,E2 -18955.018} C_VEL
LIN {X 0,Y 249.824,Z 271.149,A -85,B 0,C 180,E1 -18957.689,E2 -18957.689} C_VEL
LIN {X 0,Y 251.166,Z 263.856,A -85,B 0,C 180,E1 -18960.159,E2 -18960.159} C_VEL
LIN {X 0,Y 252.646,Z 255.965,A -85,B 0,C 180,E1 -18962.296,E2 -18962.296} C_VEL
LIN {X 0,Y 254.279,Z 246.533,A -85,B 0,C 180,E1 -18964.373,E2 -18964.373} C_VEL
LIN {X 0,Y 256.042,Z 235.455,A -85,B 0,C 180,E1 -18966.332,E2 -18966.332} C_VEL
LIN {X 0,Y 257.723,Z 223.413,A -85,B 0,C 180,E1 -18967.995,E2 -18967.995} C_VEL
LIN {X 0,Y 255.732,Z 212.221,A -85,B 0,C 180,E1 -18969.488,E2 -18969.488} C_VEL
LIN {X 0,Y 252.62,Z 199.475,A -85,B 0,C 180,E1 -18970.924,E2 -18970.924} C_VEL
LIN {X 0,Y 248.815,Z 186.618,A -85,B 0,C 180,E1 -18972.111,E2 -18972.111} C_VEL
LIN {X 0,Y 248.297,Z 184.504,A -85,B 0,C 180,E1 -18972.285,E2 -18972.285} C_VEL
LIN {X 0,Y 248.494,Z 182.259,A -85,B 0,C 180,E1 -18975.253,E2 -18975.253} C_VEL
LIN {X 0,Y 248.657,Z 181.511,A -85,B 0,C 180,E1 -18976.931,E2 -18976.931} C_VEL
LIN {X 0,Y 249.238,Z 181.438,A -85,B 0,C 180,E1 -18980.72,E2 -18980.72} C_VEL
LIN {X 0,Y 249.432,Z 181.415,A -85,B 0,C 180,E1 -18983.528,E2 -18983.528} C_VEL
LIN {X 0,Y 249.673,Z 181.385,A -85,B 0,C 180,E1 -18988.387,E2 -18988.387} C_VEL
LIN {X 0,Y 249.673,Z 181.383,A -85,B 0,C 180,E1 -18991.613,E2 -18991.613} C_VEL
LIN {X 0,Y 249.458,Z 181.411,A -85,B 0,C 180,E1 -18996.47,E2 -18996.47} C_VEL
LIN {X 0,Y 249.421,Z 181.417,A -85,B 0,C 180,E1 -18999.733,E2 -18999.733} C_VEL
LIN {X 0,Y 249.202,Z 181.444,A -85,B 0,C 180,E1 -19004.703,E2 -19004.703} C_VEL
LIN {X 0,Y 249.137,Z 181.45,A -85,B 0,C 180,E1 -19008.077,E2 -19008.077} C_VEL
LIN {X 0,Y 249.101,Z 181.46,A -85,B 0,C 180,E1 -19011.517,E2 -19011.517} C_VEL
LIN {X 0,Y 249.127,Z 181.451,A -85,B 0,C 180,E1 -19015.482,E2 -19015.482} C_VEL
LIN {X 0,Y 249.07,Z 181.458,A -85,B 0,C 180,E1 -19018.989,E2 -19018.989} C_VEL
LIN {X 0,Y 249.027,Z 181.464,A -85,B 0,C 180,E1 -19022.426,E2 -19022.426} C_VEL
LIN {X 0,Y 249.026,Z 181.457,A -85,B 0,C 180,E1 -19026.346,E2 -19026.346} C_VEL
LIN {X 0,Y 249.003,Z 181.466,A -85,B 0,C 180,E1 -19030.478,E2 -19030.478} C_VEL
LIN {X 0,Y 249.005,Z 181.468,A -85,B 0,C 180,E1 -19034.879,E2 -19034.879} C_VEL
LIN {X 0,Y 249.015,Z 181.458,A -85,B 0,C 180,E1 -19037.364,E2 -19037.364} C_VEL
LIN {X 0,Y 249.041,Z 181.46,A -85,B 0,C 180,E1 -19042.201,E2 -19042.201} C_VEL
LIN {X 0,Y 249.041,Z 181.461,A -85,B 0,C 180,E1 -19045.64,E2 -19045.64} C_VEL
LIN {X 0,Y 249.046,Z 181.455,A -85,B 0,C 180,E1 -19049.473,E2 -19049.473} C_VEL
LIN {X 0,Y 249.07,Z 181.454,A -85,B 0,C 180,E1 -19053.163,E2 -19053.163} C_VEL
LIN {X 0,Y 249.083,Z 181.458,A -85,B 0,C 180,E1 -19056.734,E2 -19056.734} C_VEL
LIN {X 0,Y 249.129,Z 181.452,A -85,B 0,C 180,E1 -19060.214,E2 -19060.214} C_VEL
LIN {X 0,Y 249.242,Z 181.429,A -85,B 0,C 180,E1 -19063.623,E2 -19063.623} C_VEL
LIN {X 0,Y 249.245,Z 181.437,A -85,B 0,C 180,E1 -19068.617,E2 -19068.617} C_VEL
LIN {X 0,Y 249.455,Z 181.412,A -85,B 0,C 180,E1 -19071.903,E2 -19071.903} C_VEL
LIN {X 0,Y 249.298,Z 181.426,A -85,B 0,C 180,E1 -19075.149,E2 -19075.149} C_VEL
LIN {X 0,Y 249.677,Z 181.38,A -85,B 0,C 180,E1 -19078.388,E2 -19078.388} C_VEL
LIN {X 0,Y 249.676,Z 181.382,A -85,B 0,C 180,E1 -19081.614,E2 -19081.614} C_VEL
LIN {X 0,Y 249.438,Z 181.41,A -85,B 0,C 180,E1 -19086.472,E2 -19086.472} C_VEL
LIN {X 0,Y 249.344,Z 181.421,A -85,B 0,C 180,E1 -19089.737,E2 -19089.737} C_VEL
LIN {X 0,Y 249.207,Z 181.441,A -85,B 0,C 180,E1 -19094.704,E2 -19094.704} C_VEL
LIN {X 0,Y 249.142,Z 181.447,A -85,B 0,C 180,E1 -19098.078,E2 -19098.078} C_VEL
LIN {X 0,Y 249.106,Z 181.457,A -85,B 0,C 180,E1 -19101.517,E2 -19101.517} C_VEL
LIN {X 0,Y 249.132,Z 181.454,A -85,B 0,C 180,E1 -19105.483,E2 -19105.483} C_VEL
LIN {X 0,Y 249.075,Z 181.46,A -85,B 0,C 180,E1 -19108.99,E2 -19108.99} C_VEL
LIN {X 0,Y 249.033,Z 181.464,A -85,B 0,C 180,E1 -19112.426,E2 -19112.426} C_VEL
LIN {X 0,Y 249.127,Z 181.493,A -85,B 0,C 180,E1 -19117.196,E2 -19117.196} C_VEL
LIN {X 0,Y 249.394,Z 183.356,A -85,B 0,C 180,E1 -19119.04,E2 -19119.04} C_VEL
LIN {X 0,Y 248.96,Z 184.828,A -85,B 0,C 180,E1 -19120.35,E2 -19120.35} C_VEL
LIN {X 0,Y 246.5,Z 187.565,A -85,B 0,C 180,E1 -19122.482,E2 -19122.482} C_VEL
LIN {X 0,Y 244.434,Z 189.808,A -85,B 0,C 180,E1 -19124.212,E2 -19124.212} C_VEL
LIN {X 0,Y 243.71,Z 191.415,A -85,B 0,C 180,E1 -19125.551,E2 -19125.551} C_VEL
LIN {X 0,Y 243.742,Z 191.92,A -85,B 0,C 180,E1 -19126.004,E2 -19126.004} C_VEL
LIN {X 0,Y 244.541,Z 196.109,A -85,B 0,C 180,E1 -19129.712,E2 -19129.712} C_VEL
LIN {X 0,Y 244.837,Z 198.719,A -85,B 0,C 180,E1 -19131.901,E2 -19131.901} C_VEL
LIN {X 0,Y 244.447,Z 202.467,A -85,B 0,C 180,E1 -19134.9,E2 -19134.9} C_VEL
LIN {X 0,Y 243.108,Z 208.498,A -85,B 0,C 180,E1 -19139.536,E2 -19139.536} C_VEL
LIN {X 0,Y 242.539,Z 211.302,A -85,B 0,C 180,E1 -19141.653,E2 -19141.653} C_VEL
LIN {X 0,Y 244.876,Z 224.96,A -85,B 0,C 180,E1 -19142.665,E2 -19142.665} C_VEL
LIN {X 0,Y 246.687,Z 237.975,A -85,B 0,C 180,E1 -19143.94,E2 -19143.94} C_VEL
LIN {X 0,Y 247.816,Z 250.059,A -85,B 0,C 180,E1 -19145.407,E2 -19145.407} C_VEL
LIN {X 0,Y 248.351,Z 261.574,A -85,B 0,C 180,E1 -19147.101,E2 -19147.101} C_VEL
LIN {X 0,Y 248.366,Z 265.534,A -85,B 0,C 180,E1 -19147.761,E2 -19147.761} C_VEL
LIN {X 0,Y 246.52,Z 275.453,A -85,B 0,C 180,E1 -19149.56,E2 -19149.56} C_VEL
LIN {X 0,Y 244.779,Z 284.484,A -85,B 0,C 180,E1 -19151.589,E2 -19151.589} C_VEL
LIN {X 0,Y 243.338,Z 291.967,A -85,B 0,C 180,E1 -19153.645,E2 -19153.645} C_VEL
LIN {X 0,Y 241.946,Z 299.318,A -85,B 0,C 180,E1 -19156.135,E2 -19156.135} C_VEL
LIN {X 0,Y 240.874,Z 306.061,A -85,B 0,C 180,E1 -19159.068,E2 -19159.068} C_VEL
LIN {X 0,Y 240.343,Z 310.493,A -85,B 0,C 180,E1 -19161.593,E2 -19161.593} C_VEL
LIN {X 0,Y 240.096,Z 314.129,A -85,B 0,C 180,E1 -19164.413,E2 -19164.413} C_VEL
LIN {X 0,Y 240.057,Z 316.131,A -85,B 0,C 180,E1 -19166.644,E2 -19166.644} C_VEL
LIN {X 0,Y 240.037,Z 317.109,A -85,B 0,C 180,E1 -19168.322,E2 -19168.322} C_VEL
LIN {X 0,Y 240.097,Z 317.688,A -85,B 0,C 180,E1 -19170,E2 -19170} C_VEL
LIN {X 0,Y 240.024,Z 317.859,A -85,B 0,C 180,E1 -19171.678,E2 -19171.678} C_VEL
LIN {X 0,Y 239.981,Z 317.604,A -85,B 0,C 180,E1 -19173.358,E2 -19173.358} C_VEL
LIN {X 0,Y 240.078,Z 315.875,A -85,B 0,C 180,E1 -19176.725,E2 -19176.725} C_VEL
LIN {X 0,Y 240.248,Z 314.424,A -85,B 0,C 180,E1 -19178.411,E2 -19178.411} C_VEL
LIN {X 0,Y 240.855,Z 311.437,A -85,B 0,C 180,E1 -19180.934,E2 -19180.934} C_VEL
LIN {X 0,Y 241.809,Z 307.452,A -85,B 0,C 180,E1 -19183.445,E2 -19183.445} C_VEL
LIN {X 0,Y 243.37,Z 302.383,A -85,B 0,C 180,E1 -19185.923,E2 -19185.923} C_VEL
LIN {X 0,Y 245.259,Z 296.086,A -85,B 0,C 180,E1 -19188.374,E2 -19188.374} C_VEL
LIN {X 0,Y 247.521,Z 288.374,A -85,B 0,C 180,E1 -19190.789,E2 -19190.789} C_VEL
LIN {X 0,Y 250.281,Z 278.84,A -85,B 0,C 180,E1 -19193.15,E2 -19193.15} C_VEL
LIN {X 0,Y 252.626,Z 270.188,A -85,B 0,C 180,E1 -19194.884,E2 -19194.884} C_VEL
LIN {X 0,Y 253.638,Z 258.529,A -85,B 0,C 180,E1 -19197.021,E2 -19197.021} C_VEL
LIN {X 0,Y 253.563,Z 248.349,A -85,B 0,C 180,E1 -19198.678,E2 -19198.678} C_VEL
LIN {X 0,Y 252.48,Z 237.297,A -85,B 0,C 180,E1 -19200.353,E2 -19200.353} C_VEL
LIN {X 0,Y 250.364,Z 226.556,A -85,B 0,C 180,E1 -19201.92,E2 -19201.92} C_VEL
LIN {X 0,Y 247.148,Z 215.286,A -85,B 0,C 180,E1 -19203.556,E2 -19203.556} C_VEL
LIN {X 0,Y 245.745,Z 211.11,A -85,B 0,C 180,E1 -19204.155,E2 -19204.155} C_VEL
LIN {X 0,Y 244.774,Z 207.589,A -85,B 0,C 180,E1 -19204.615,E2 -19204.615} C_VEL
LIN {X 0,Y 245.494,Z 203.789,A -85,B 0,C 180,E1 -19207.989,E2 -19207.989} C_VEL
LIN {X 0,Y 245.263,Z 200.56,A -85,B 0,C 180,E1 -19211.229,E2 -19211.229} C_VEL
LIN {X 0,Y 244.498,Z 196.422,A -85,B 0,C 180,E1 -19215.941,E2 -19215.941} C_VEL
LIN {X 0,Y 243.882,Z 192.873,A -85,B 0,C 180,E1 -19220.655,E2 -19220.655} C_VEL
LIN {X 0,Y 243.448,Z 190.274,A -85,B 0,C 180,E1 -19224.733,E2 -19224.733} C_VEL
LIN {X 0,Y 243.073,Z 188.23,A -85,B 0,C 180,E1 -19228.638,E2 -19228.638} C_VEL
LIN {X 0,Y 242.837,Z 186.639,A -85,B 0,C 180,E1 -19232.414,E2 -19232.414} C_VEL
LIN {X 0,Y 242.628,Z 185.489,A -85,B 0,C 180,E1 -19236.075,E2 -19236.075} C_VEL
LIN {X 0,Y 242.507,Z 184.7,A -85,B 0,C 180,E1 -19239.648,E2 -19239.648} C_VEL
LIN {X 0,Y 242.471,Z 184.239,A -85,B 0,C 180,E1 -19243.15,E2 -19243.15} C_VEL
LIN {X 0,Y 242.488,Z 184.081,A -85,B 0,C 180,E1 -19246.592,E2 -19246.592} C_VEL
LIN {X 0,Y 242.686,Z 184.167,A -85,B 0,C 180,E1 -19249.993,E2 -19249.993} C_VEL
LIN {X 0,Y 242.798,Z 184.537,A -85,B 0,C 180,E1 -19253.35,E2 -19253.35} C_VEL
LIN {X 0,Y 243.167,Z 185.484,A -85,B 0,C 180,E1 -19258.343,E2 -19258.343} C_VEL
LIN {X 0,Y 243.333,Z 185.9,A -85,B 0,C 180,E1 -19259.999,E2 -19259.999} C_VEL
LIN {X 0,Y 243.206,Z 186.982,A -85,B 0,C 180,E1 -19263.312,E2 -19263.312} C_VEL
LIN {X 0,Y 243.261,Z 188.241,A -85,B 0,C 180,E1 -19266.729,E2 -19266.729} C_VEL
LIN {X 0,Y 243.171,Z 189.962,A -85,B 0,C 180,E1 -19270.244,E2 -19270.244} C_VEL
LIN {X 0,Y 244.314,Z 192.946,A -85,B 0,C 180,E1 -19270.739,E2 -19270.739} C_VEL
LIN {X 0,Y 245.476,Z 194.709,A -85,B 0,C 180,E1 -19271.135,E2 -19271.135} C_VEL
LIN {X 0,Y 249.996,Z 204.338,A -85,B 0,C 180,E1 -19272.996,E2 -19272.996} C_VEL
LIN {X 0,Y 254.173,Z 215.573,A -85,B 0,C 180,E1 -19275.105,E2 -19275.105} C_VEL
LIN {X 0,Y 256.56,Z 225.31,A -85,B 0,C 180,E1 -19276.92,E2 -19276.92} C_VEL
LIN {X 0,Y 257.945,Z 234.396,A -85,B 0,C 180,E1 -19278.671,E2 -19278.671} C_VEL
LIN {X 0,Y 255.167,Z 245.672,A -85,B 0,C 180,E1 -19280.535,E2 -19280.535} C_VEL
LIN {X 0,Y 252.63,Z 255.012,A -85,B 0,C 180,E1 -19282.489,E2 -19282.489} C_VEL
LIN {X 0,Y 250.295,Z 262.681,A -85,B 0,C 180,E1 -19284.465,E2 -19284.465} C_VEL
LIN {X 0,Y 247.732,Z 270.526,A -85,B 0,C 180,E1 -19286.994,E2 -19286.994} C_VEL
LIN {X 0,Y 245.311,Z 277.267,A -85,B 0,C 180,E1 -19289.807,E2 -19289.807} C_VEL
LIN {X 0,Y 243.742,Z 281.505,A -85,B 0,C 180,E1 -19292.122,E2 -19292.122} C_VEL
LIN {X 0,Y 242.567,Z 284.699,A -85,B 0,C 180,E1 -19294.4,E2 -19294.4} C_VEL
LIN {X 0,Y 241.179,Z 287.892,A -85,B 0,C 180,E1 -19297.729,E2 -19297.729} C_VEL
LIN {X 0,Y 240.438,Z 289.265,A -85,B 0,C 180,E1 -19300.537,E2 -19300.537} C_VEL
LIN {X 0,Y 240.092,Z 289.555,A -85,B 0,C 180,E1 -19302.962,E2 -19302.962} C_VEL
LIN {X 0,Y 239.934,Z 289.005,A -85,B 0,C 180,E1 -19305.332,E2 -19305.332} C_VEL
LIN {X 0,Y 240.021,Z 287.689,A -85,B 0,C 180,E1 -19307.665,E2 -19307.665} C_VEL
LIN {X 0,Y 240.349,Z 285.62,A -85,B 0,C 180,E1 -19309.961,E2 -19309.961} C_VEL
LIN {X 0,Y 240.846,Z 282.81,A -85,B 0,C 180,E1 -19312.208,E2 -19312.208} C_VEL
LIN {X 0,Y 241.502,Z 278.912,A -85,B 0,C 180,E1 -19314.569,E2 -19314.569} C_VEL
LIN {X 0,Y 242.488,Z 273.35,A -85,B 0,C 180,E1 -19317.192,E2 -19317.192} C_VEL
LIN {X 0,Y 243.836,Z 266.131,A -85,B 0,C 180,E1 -19319.844,E2 -19319.844} C_VEL
LIN {X 0,Y 245.39,Z 258.266,A -85,B 0,C 180,E1 -19322.154,E2 -19322.154} C_VEL
LIN {X 0,Y 247.03,Z 249.319,A -85,B 0,C 180,E1 -19324.287,E2 -19324.287} C_VEL
LIN {X 0,Y 248.691,Z 239.061,A -85,B 0,C 180,E1 -19326.252,E2 -19326.252} C_VEL
LIN {X 0,Y 250.491,Z 227.627,A -85,B 0,C 180,E1 -19327.996,E2 -19327.996} C_VEL
LIN {X 0,Y 250.935,Z 224.43,A -85,B 0,C 180,E1 -19328.411,E2 -19328.411} C_VEL
LIN {X 0,Y 248.892,Z 213.158,A -85,B 0,C 180,E1 -19329.978,E2 -19329.978} C_VEL
LIN {X 0,Y 245.808,Z 200.619,A -85,B 0,C 180,E1 -19331.453,E2 -19331.453} C_VEL
LIN {X 0,Y 242.084,Z 187.802,A -85,B 0,C 180,E1 -19332.688,E2 -19332.688} C_VEL
LIN {X 0,Y 241.288,Z 184.895,A -85,B 0,C 180,E1 -19332.957,E2 -19332.957} C_VEL
LIN {X 0,Y 241.531,Z 182.401,A -85,B 0,C 180,E1 -19336.539,E2 -19336.539} C_VEL
LIN {X 0,Y 242.187,Z 182.317,A -85,B 0,C 180,E1 -19340.619,E2 -19340.619} C_VEL
LIN {X 0,Y 242.395,Z 182.291,A -85,B 0,C 180,E1 -19343.34,E2 -19343.34} C_VEL
LIN {X 0,Y 242.634,Z 182.263,A -85,B 0,C 180,E1 -19348.34,E2 -19348.34} C_VEL
LIN {X 0,Y 242.634,Z 182.26,A -85,B 0,C 180,E1 -19351.66,E2 -19351.66} C_VEL
LIN {X 0,Y 242.431,Z 182.286,A -85,B 0,C 180,E1 -19356.659,E2 -19356.659} C_VEL
LIN {X 0,Y 242.342,Z 182.296,A -85,B 0,C 180,E1 -19360.02,E2 -19360.02} C_VEL
LIN {X 0,Y 242.164,Z 182.322,A -85,B 0,C 180,E1 -19365.141,E2 -19365.141} C_VEL
LIN {X 0,Y 242.076,Z 182.328,A -85,B 0,C 180,E1 -19368.624,E2 -19368.624} C_VEL
LIN {X 0,Y 242.047,Z 182.336,A -85,B 0,C 180,E1 -19372.176,E2 -19372.176} C_VEL
LIN {X 0,Y 242.063,Z 182.327,A -85,B 0,C 180,E1 -19375.838,E2 -19375.838} C_VEL
LIN {X 0,Y 242.004,Z 182.342,A -85,B 0,C 180,E1 -19379.583,E2 -19379.583} C_VEL
LIN {X 0,Y 241.977,Z 182.342,A -85,B 0,C 180,E1 -19383.493,E2 -19383.493} C_VEL
LIN {X 0,Y 241.983,Z 182.338,A -85,B 0,C 180,E1 -19387.583,E2 -19387.583} C_VEL
LIN {X 0,Y 241.936,Z 182.347,A -85,B 0,C 180,E1 -19391.922,E2 -19391.922} C_VEL
LIN {X 0,Y 241.934,Z 182.344,A -85,B 0,C 180,E1 -19396.571,E2 -19396.571} C_VEL
LIN {X 0,Y 241.954,Z 182.34,A -85,B 0,C 180,E1 -19400.282,E2 -19400.282} C_VEL
LIN {X 0,Y 241.979,Z 182.342,A -85,B 0,C 180,E1 -19404.489,E2 -19404.489} C_VEL
LIN {X 0,Y 241.972,Z 182.342,A -85,B 0,C 180,E1 -19408.48,E2 -19408.48} C_VEL
LIN {X 0,Y 242.001,Z 182.331,A -85,B 0,C 180,E1 -19412.313,E2 -19412.313} C_VEL
LIN {X 0,Y 242.059,Z 182.33,A -85,B 0,C 180,E1 -19416.017,E2 -19416.017} C_VEL
LIN {X 0,Y 242.06,Z 182.33,A -85,B 0,C 180,E1 -19419.611,E2 -19419.611} C_VEL
LIN {X 0,Y 242.163,Z 182.311,A -85,B 0,C 180,E1 -19423.279,E2 -19423.279} C_VEL
LIN {X 0,Y 242.181,Z 182.316,A -85,B 0,C 180,E1 -19428.28,E2 -19428.28} C_VEL
LIN {X 0,Y 242.401,Z 182.289,A -85,B 0,C 180,E1 -19431.666,E2 -19431.666} C_VEL
LIN {X 0,Y 242.259,Z 182.302,A -85,B 0,C 180,E1 -19435.008,E2 -19435.008} C_VEL
LIN {X 0,Y 242.637,Z 182.256,A -85,B 0,C 180,E1 -19438.341,E2 -19438.341} C_VEL
LIN {X 0,Y 242.636,Z 182.26,A -85,B 0,C 180,E1 -19441.661,E2 -19441.661} C_VEL
LIN {X 0,Y 242.409,Z 182.285,A -85,B 0,C 180,E1 -19446.66,E2 -19446.66} C_VEL
LIN {X 0,Y 242.269,Z 182.304,A -85,B 0,C 180,E1 -19450.025,E2 -19450.025} C_VEL
LIN {X 0,Y 242.168,Z 182.318,A -85,B 0,C 180,E1 -19455.142,E2 -19455.142} C_VEL
LIN {X 0,Y 242.081,Z 182.325,A -85,B 0,C 180,E1 -19458.624,E2 -19458.624} C_VEL
LIN {X 0,Y 242.052,Z 182.333,A -85,B 0,C 180,E1 -19462.177,E2 -19462.177} C_VEL
LIN {X 0,Y 242.069,Z 182.333,A -85,B 0,C 180,E1 -19465.839,E2 -19465.839} C_VEL
LIN {X 0,Y 242.009,Z 182.341,A -85,B 0,C 180,E1 -19469.584,E2 -19469.584} C_VEL
LIN {X 0,Y 241.983,Z 182.344,A -85,B 0,C 180,E1 -19473.493,E2 -19473.493} C_VEL
LIN {X 0,Y 242.063,Z 182.421,A -85,B 0,C 180,E1 -19476.786,E2 -19476.786} C_VEL
LIN {X 0,Y 242.805,Z 186.804,A -85,B 0,C 180,E1 -19481.187,E2 -19481.187} C_VEL
LIN {X 0,Y 243.521,Z 190.823,A -85,B 0,C 180,E1 -19484.998,E2 -19484.998} C_VEL
LIN {X 0,Y 243.742,Z 191.92,A -85,B 0,C 180,E1 -19486.004,E2 -19486.004} C_VEL
LIN {X 0,Y 243.445,Z 193.488,A -85,B 0,C 180,E1 -19487.339,E2 -19487.339} C_VEL
LIN {X 0,Y 242.227,Z 195.183,A -85,B 0,C 180,E1 -19488.65,E2 -19488.65} C_VEL
LIN {X 0,Y 238.14,Z 199.873,A -85,B 0,C 180,E1 -19492.179,E2 -19492.179} C_VEL
LIN {X 0,Y 237.712,Z 201.016,A -85,B 0,C 180,E1 -19493.099,E2 -19493.099} C_VEL
LIN {X 0,Y 236.942,Z 204.783,A -85,B 0,C 180,E1 -19496.153,E2 -19496.153} C_VEL
LIN {X 0,Y 235.614,Z 210.905,A -85,B 0,C 180,E1 -19500.96,E2 -19500.96} C_VEL
LIN {X 0,Y 237.956,Z 224.817,A -85,B 0,C 180,E1 -19502.044,E2 -19502.044} C_VEL
LIN {X 0,Y 239.775,Z 238.167,A -85,B 0,C 180,E1 -19503.411,E2 -19503.411} C_VEL
LIN {X 0,Y 240.949,Z 251.077,A -85,B 0,C 180,E1 -19505.047,E2 -19505.047} C_VEL
LIN {X 0,Y 241.434,Z 262.708,A -85,B 0,C 180,E1 -19506.86,E2 -19506.86} C_VEL
LIN {X 0,Y 241.28,Z 266.54,A -85,B 0,C 180,E1 -19507.524,E2 -19507.524} C_VEL
LIN {X 0,Y 239.424,Z 276.199,A -85,B 0,C 180,E1 -19509.375,E2 -19509.375} C_VEL
LIN {X 0,Y 237.68,Z 285.042,A -85,B 0,C 180,E1 -19511.466,E2 -19511.466} C_VEL
LIN {X 0,Y 236.21,Z 292.36,A -85,B 0,C 180,E1 -19513.582,E2 -19513.582} C_VEL
LIN {X 0,Y 234.794,Z 299.563,A -85,B 0,C 180,E1 -19516.146,E2 -19516.146} C_VEL
LIN {X 0,Y 233.879,Z 305.313,A -85,B 0,C 180,E1 -19518.737,E2 -19518.737} C_VEL
LIN {X 0,Y 233.286,Z 309.816,A -85,B 0,C 180,E1 -19521.337,E2 -19521.337} C_VEL
LIN {X 0,Y 233.032,Z 313.703,A -85,B 0,C 180,E1 -19524.419,E2 -19524.419} C_VEL
LIN {X 0,Y 232.973,Z 315.584,A -85,B 0,C 180,E1 -19526.541,E2 -19526.541} C_VEL
LIN {X 0,Y 232.967,Z 316.599,A -85,B 0,C 180,E1 -19528.272,E2 -19528.272} C_VEL
LIN {X 0,Y 233.021,Z 317.209,A -85,B 0,C 180,E1 -19530,E2 -19530} C_VEL
LIN {X 0,Y 232.952,Z 317.412,A -85,B 0,C 180,E1 -19531.729,E2 -19531.729} C_VEL
LIN {X 0,Y 232.895,Z 317.215,A -85,B 0,C 180,E1 -19533.46,E2 -19533.46} C_VEL
LIN {X 0,Y 233.002,Z 315.561,A -85,B 0,C 180,E1 -19536.93,E2 -19536.93} C_VEL
LIN {X 0,Y 233.594,Z 312.328,A -85,B 0,C 180,E1 -19540.4,E2 -19540.4} C_VEL
LIN {X 0,Y 234.504,Z 308.753,A -85,B 0,C 180,E1 -19542.99,E2 -19542.99} C_VEL
LIN {X 0,Y 235.939,Z 304.156,A -85,B 0,C 180,E1 -19545.551,E2 -19545.551} C_VEL
LIN {X 0,Y 238.128,Z 297.311,A -85,B 0,C 180,E1 -19548.498,E2 -19548.498} C_VEL
LIN {X 0,Y 240.475,Z 289.968,A -85,B 0,C 180,E1 -19550.979,E2 -19550.979} C_VEL
LIN {X 0,Y 243.27,Z 280.976,A -85,B 0,C 180,E1 -19553.406,E2 -19553.406} C_VEL
LIN {X 0,Y 246.047,Z 271.808,A -85,B 0,C 180,E1 -19555.37,E2 -19555.37} C_VEL
LIN {X 0,Y 247.313,Z 259.617,A -85,B 0,C 180,E1 -19557.739,E2 -19557.739} C_VEL
LIN {X 0,Y 247.384,Z 249.545,A -85,B 0,C 180,E1 -19559.484,E2 -19559.484} C_VEL
LIN {X 0,Y 246.28,Z 237.78,A -85,B 0,C 180,E1 -19561.386,E2 -19561.386} C_VEL
LIN {X 0,Y 244.142,Z 226.446,A -85,B 0,C 180,E1 -19563.158,E2 -19563.158} C_VEL
LIN {X 0,Y 240.884,Z 215.101,A -85,B 0,C 180,E1 -19564.931,E2 -19564.931} C_VEL
LIN {X 0,Y 239.545,Z 211.317,A -85,B 0,C 180,E1 -19565.535,E2 -19565.535} C_VEL
LIN {X 0,Y 238.308,Z 208.078,A -85,B 0,C 180,E1 -19566.072,E2 -19566.072} C_VEL
LIN {X 0,Y 238.158,Z 206.942,A -85,B 0,C 180,E1 -19566.241,E2 -19566.241} C_VEL
LIN {X 0,Y 238.506,Z 204.822,A -85,B 0,C 180,E1 -19568.229,E2 -19568.229} C_VEL
LIN {X 0,Y 238.368,Z 202.67,A -85,B 0,C 180,E1 -19570.44,E2 -19570.44} C_VEL
LIN {X 0,Y 238.033,Z 200.567,A -85,B 0,C 180,E1 -19572.773,E2 -19572.773} C_VEL
LIN {X 0,Y 237.36,Z 197.05,A -85,B 0,C 180,E1 -19577.076,E2 -19577.076} C_VEL
LIN {X 0,Y 236.876,Z 193.934,A -85,B 0,C 180,E1 -19581.459,E2 -19581.459} C_VEL
LIN {X 0,Y 236.421,Z 191.472,A -85,B 0,C 180,E1 -19585.61,E2 -19585.61} C_VEL
LIN {X 0,Y 236.099,Z 189.478,A -85,B 0,C 180,E1 -19589.684,E2 -19589.684} C_VEL
LIN {X 0,Y 235.893,Z 188.019,A -85,B 0,C 180,E1 -19593.454,E2 -19593.454} C_VEL
LIN {X 0,Y 235.667,Z 186.87,A -85,B 0,C 180,E1 -19597.59,E2 -19597.59} C_VEL
LIN {X 0,Y 235.596,Z 186.021,A -85,B 0,C 180,E1 -19602.668,E2 -19602.668} C_VEL
LIN {X 0,Y 235.604,Z 185.803,A -85,B 0,C 180,E1 -19606.193,E2 -19606.193} C_VEL
LIN {X 0,Y 235.768,Z 185.846,A -85,B 0,C 180,E1 -19609.696,E2 -19609.696} C_VEL
LIN {X 0,Y 235.88,Z 186.167,A -85,B 0,C 180,E1 -19613.154,E2 -19613.154} C_VEL
LIN {X 0,Y 236.248,Z 187.058,A -85,B 0,C 180,E1 -19618.294,E2 -19618.294} C_VEL
LIN {X 0,Y 236.408,Z 187.458,A -85,B 0,C 180,E1 -19619.999,E2 -19619.999} C_VEL
LIN {X 0,Y 236.258,Z 188.52,A -85,B 0,C 180,E1 -19623.41,E2 -19623.41} C_VEL
LIN {X 0,Y 236.281,Z 190.077,A -85,B 0,C 180,E1 -19627.691,E2 -19627.691} C_VEL
LIN {X 0,Y 236.286,Z 190.59,A -85,B 0,C 180,E1 -19628.552,E2 -19628.552} C_VEL
LIN {X 0,Y 237.362,Z 193.32,A -85,B 0,C 180,E1 -19629.049,E2 -19629.049} C_VEL
LIN {X 0,Y 238.918,Z 195.539,A -85,B 0,C 180,E1 -19629.63,E2 -19629.63} C_VEL
LIN {X 0,Y 244.357,Z 207.029,A -85,B 0,C 180,E1 -19632.072,E2 -19632.072} C_VEL
LIN {X 0,Y 247.752,Z 216.427,A -85,B 0,C 180,E1 -19633.976,E2 -19633.976} C_VEL
LIN {X 0,Y 250.249,Z 226.016,A -85,B 0,C 180,E1 -19635.891,E2 -19635.891} C_VEL
LIN {X 0,Y 251.677,Z 235.767,A -85,B 0,C 180,E1 -19637.888,E2 -19637.888} C_VEL
LIN {X 0,Y 250.988,Z 239.402,A -85,B 0,C 180,E1 -19638.498,E2 -19638.498} C_VEL
LIN {X 0,Y 248.389,Z 248.91,A -85,B 0,C 180,E1 -19640.224,E2 -19640.224} C_VEL
LIN {X 0,Y 245.447,Z 258.668,A -85,B 0,C 180,E1 -19642.464,E2 -19642.464} C_VEL
LIN {X 0,Y 242.781,Z 266.619,A -85,B 0,C 180,E1 -19644.752,E2 -19644.752} C_VEL
LIN {X 0,Y 240.156,Z 273.92,A -85,B 0,C 180,E1 -19647.445,E2 -19647.445} C_VEL
LIN {X 0,Y 237.981,Z 279.547,A -85,B 0,C 180,E1 -19650.134,E2 -19650.134} C_VEL
LIN {X 0,Y 236.527,Z 283.133,A -85,B 0,C 180,E1 -19652.332,E2 -19652.332} C_VEL
LIN {X 0,Y 235.394,Z 285.935,A -85,B 0,C 180,E1 -19654.559,E2 -19654.559} C_VEL
LIN {X 0,Y 234.42,Z 287.987,A -85,B 0,C 180,E1 -19656.841,E2 -19656.841} C_VEL
LIN {X 0,Y 233.67,Z 289.335,A -85,B 0,C 180,E1 -19659.168,E2 -19659.168} C_VEL
LIN {X 0,Y 233.197,Z 289.969,A -85,B 0,C 180,E1 -19661.53,E2 -19661.53} C_VEL
LIN {X 0,Y 232.924,Z 289.823,A -85,B 0,C 180,E1 -19663.945,E2 -19663.945} C_VEL
LIN {X 0,Y 232.86,Z 288.861,A -85,B 0,C 180,E1 -19666.413,E2 -19666.413} C_VEL
LIN {X 0,Y 233.065,Z 287.036,A -85,B 0,C 180,E1 -19668.925,E2 -19668.925} C_VEL
LIN {X 0,Y 233.568,Z 284.262,A -85,B 0,C 180,E1 -19671.473,E2 -19671.473} C_VEL
LIN {X 0,Y 234.257,Z 280.351,A -85,B 0,C 180,E1 -19674.097,E2 -19674.097} C_VEL
LIN {X 0,Y 235.223,Z 275.116,A -85,B 0,C 180,E1 -19676.78,E2 -19676.78} C_VEL
LIN {X 0,Y 236.598,Z 267.862,A -85,B 0,C 180,E1 -19679.67,E2 -19679.67} C_VEL
LIN {X 0,Y 238.264,Z 259.582,A -85,B 0,C 180,E1 -19682.237,E2 -19682.237} C_VEL
LIN {X 0,Y 239.975,Z 250.511,A -85,B 0,C 180,E1 -19684.504,E2 -19684.504} C_VEL
LIN {X 0,Y 241.648,Z 241.087,A -85,B 0,C 180,E1 -19686.412,E2 -19686.412} C_VEL
LIN {X 0,Y 243.543,Z 229.437,A -85,B 0,C 180,E1 -19688.287,E2 -19688.287} C_VEL
LIN {X 0,Y 244.099,Z 225.583,A -85,B 0,C 180,E1 -19688.818,E2 -19688.818} C_VEL
LIN {X 0,Y 241.99,Z 214.051,A -85,B 0,C 180,E1 -19690.489,E2 -19690.489} C_VEL
LIN {X 0,Y 239.148,Z 202.146,A -85,B 0,C 180,E1 -19691.96,E2 -19691.96} C_VEL
LIN {X 0,Y 235.622,Z 189.964,A -85,B 0,C 180,E1 -19693.216,E2 -19693.216} C_VEL
LIN {X 0,Y 234.296,Z 185.302,A -85,B 0,C 180,E1 -19693.65,E2 -19693.65} C_VEL
LIN {X 0,Y 234.432,Z 183.539,A -85,B 0,C 180,E1 -19696.123,E2 -19696.123} C_VEL
LIN {X 0,Y 235.12,Z 183.198,A -85,B 0,C 180,E1 -19700.536,E2 -19700.536} C_VEL
LIN {X 0,Y 235.334,Z 183.171,A -85,B 0,C 180,E1 -19703.139,E2 -19703.139} C_VEL
LIN {X 0,Y 235.593,Z 183.14,A -85,B 0,C 180,E1 -19708.29,E2 -19708.29} C_VEL
LIN {X 0,Y 235.594,Z 183.137,A -85,B 0,C 180,E1 -19711.709,E2 -19711.709} C_VEL
LIN {X 0,Y 235.403,Z 183.162,A -85,B 0,C 180,E1 -19716.858,E2 -19716.858} C_VEL
LIN {X 0,Y 235.25,Z 183.178,A -85,B 0,C 180,E1 -19720.326,E2 -19720.326} C_VEL
LIN {X 0,Y 235.111,Z 183.202,A -85,B 0,C 180,E1 -19725.606,E2 -19725.606} C_VEL
LIN {X 0,Y 235.017,Z 183.209,A -85,B 0,C 180,E1 -19729.205,E2 -19729.205} C_VEL
LIN {X 0,Y 234.978,Z 183.217,A -85,B 0,C 180,E1 -19732.881,E2 -19732.881} C_VEL
LIN {X 0,Y 234.965,Z 183.21,A -85,B 0,C 180,E1 -19736.658,E2 -19736.658} C_VEL
LIN {X 0,Y 234.919,Z 183.222,A -85,B 0,C 180,E1 -19740.569,E2 -19740.569} C_VEL
LIN {X 0,Y 234.923,Z 183.218,A -85,B 0,C 180,E1 -19744.639,E2 -19744.639} C_VEL
LIN {X 0,Y 234.939,Z 183.217,A -85,B 0,C 180,E1 -19748.945,E2 -19748.945} C_VEL
LIN {X 0,Y 234.887,Z 183.225,A -85,B 0,C 180,E1 -19753.486,E2 -19753.486} C_VEL
LIN {X 0,Y 234.887,Z 183.221,A -85,B 0,C 180,E1 -19756.515,E2 -19756.515} C_VEL
LIN {X 0,Y 234.916,Z 183.221,A -85,B 0,C 180,E1 -19761.08,E2 -19761.08} C_VEL
LIN {X 0,Y 234.925,Z 183.22,A -85,B 0,C 180,E1 -19765.362,E2 -19765.362} C_VEL
LIN {X 0,Y 234.921,Z 183.213,A -85,B 0,C 180,E1 -19769.432,E2 -19769.432} C_VEL
LIN {X 0,Y 234.992,Z 183.207,A -85,B 0,C 180,E1 -19773.795,E2 -19773.795} C_VEL
LIN {X 0,Y 235.027,Z 183.207,A -85,B 0,C 180,E1 -19778.972,E2 -19778.972} C_VEL
LIN {X 0,Y 235.096,Z 183.191,A -85,B 0,C 180,E1 -19783.06,E2 -19783.06} C_VEL
LIN {X 0,Y 235.115,Z 183.194,A -85,B 0,C 180,E1 -19787.923,E2 -19787.923} C_VEL
LIN {X 0,Y 235.332,Z 183.169,A -85,B 0,C 180,E1 -19791.413,E2 -19791.413} C_VEL
LIN {X 0,Y 235.374,Z 183.163,A -85,B 0,C 180,E1 -19793.141,E2 -19793.141} C_VEL
LIN {X 0,Y 235.597,Z 183.131,A -85,B 0,C 180,E1 -19798.291,E2 -19798.291} C_VEL
LIN {X 0,Y 235.596,Z 183.137,A -85,B 0,C 180,E1 -19801.71,E2 -19801.71} C_VEL
LIN {X 0,Y 235.361,Z 183.162,A -85,B 0,C 180,E1 -19806.861,E2 -19806.861} C_VEL
LIN {X 0,Y 235.215,Z 183.182,A -85,B 0,C 180,E1 -19810.328,E2 -19810.328} C_VEL
LIN {X 0,Y 235.116,Z 183.199,A -85,B 0,C 180,E1 -19815.607,E2 -19815.607} C_VEL
LIN {X 0,Y 235.022,Z 183.205,A -85,B 0,C 180,E1 -19819.205,E2 -19819.205} C_VEL
LIN {X 0,Y 234.983,Z 183.213,A -85,B 0,C 180,E1 -19822.881,E2 -19822.881} C_VEL
LIN {X 0,Y 234.97,Z 183.215,A -85,B 0,C 180,E1 -19826.658,E2 -19826.658} C_VEL
LIN {X 0,Y 234.924,Z 183.221,A -85,B 0,C 180,E1 -19830.57,E2 -19830.57} C_VEL
LIN {X 0,Y 234.934,Z 183.221,A -85,B 0,C 180,E1 -19834.638,E2 -19834.638} C_VEL
LIN {X 0,Y 235.019,Z 183.327,A -85,B 0,C 180,E1 -19836.36,E2 -19836.36} C_VEL
LIN {X 0,Y 235.762,Z 187.8,A -85,B 0,C 180,E1 -19840.982,E2 -19840.982} C_VEL
LIN {X 0,Y 236.604,Z 192.414,A -85,B 0,C 180,E1 -19845.471,E2 -19845.471} C_VEL
LIN {X 0,Y 237.449,Z 196.687,A -85,B 0,C 180,E1 -19849.372,E2 -19849.372} C_VEL
LIN {X 0,Y 237.769,Z 199.274,A -85,B 0,C 180,E1 -19851.631,E2 -19851.631} C_VEL
LIN {X 0,Y 237.712,Z 201.016,A -85,B 0,C 180,E1 -19853.099,E2 -19853.099} C_VEL
LIN {X 0,Y 236.766,Z 202.73,A -85,B 0,C 180,E1 -19854.441,E2 -19854.441} C_VEL
LIN {X 0,Y 233.378,Z 205.681,A -85,B 0,C 180,E1 -19856.594,E2 -19856.594} C_VEL
LIN {X 0,Y 229.343,Z 209.262,A -85,B 0,C 180,E1 -19859.256,E2 -19859.256} C_VEL
LIN {X 0,Y 228.719,Z 210.452,A -85,B 0,C 180,E1 -19860.196,E2 -19860.196} C_VEL
LIN {X 0,Y 231.235,Z 225.659,A -85,B 0,C 180,E1 -19861.486,E2 -19861.486} C_VEL
LIN {X 0,Y 233.045,Z 239.488,A -85,B 0,C 180,E1 -19862.986,E2 -19862.986} C_VEL
LIN {X 0,Y 234.007,Z 251.097,A -85,B 0,C 180,E1 -19864.54,E2 -19864.54} C_VEL
LIN {X 0,Y 234.504,Z 262.395,A -85,B 0,C 180,E1 -19866.369,E2 -19866.369} C_VEL
